// TwinCAT 3 PLC project PLC
// ProgramVersion: 3.1.4024.0
// libraries:
//   EfficientIO Communicator, * (EfficientIO)
//   EfficientIO Energy Basic, * (EfficientIO)
//   EfficientIO ModbusTCP, * (EfficientIO)
//   Lynus Energy ModbusRTU, * (Lynus AG)
//   Lynus Persistent Data V1, * (Lynus AG)
//   Lynus Standards, * (EfficientIO)
//   Tc2_Math, * (Beckhoff Automation GmbH)
//   Tc2_MBus, * (Beckhoff Automation GmbH)
//   Tc2_Standard, * (Beckhoff Automation GmbH)
//   Tc2_System, * (Beckhoff Automation GmbH)
//   Tc2_Utilities, * (Beckhoff Automation GmbH)
//   Tc3_JsonXml, * (Beckhoff Automation GmbH)
//   Tc3_Module, * (Beckhoff Automation GmbH)
// project tree:
//   / Fast_Task.TcTTO, Middle_Task.TcTTO, Slow_Task.TcTTO (not stored)
//   FB/ FB_Delta_PV_Inverter_Sunspec.TcPOU, FB_KL6xxx_ModbusRTU_22B_Master.TcPOU (not stored), FB_Shelly_3EM.TcPOU, FB_Shelly_3EM_Helper.TcPOU, FB_Shelly_HT.TcPOU (not stored), FB_Shelly_HTplus.TcPOU, FB_Shelly_HTplus_Helper.TcPOU (not stored), FB_Shelly_HT_Helper.TcPOU (not stored)
//   POUs/Backup/ prgEM.TcPOU (not stored) (excluded from build), prgEMS.TcPOU (excluded from build), prgGrid.TcPOU (excluded from build), prgHouse.TcPOU (excluded from build), prgMBUS.TcPOU (excluded from build), prgPV.TcPOU (excluded from build)
//   POUs/ MAIN.TcPOU (not stored), prgComEffIO.TcPOU, prgUv12a.TcPOU, prgPersistent.TcPOU (not stored), prgRWEffIO.TcPOU (not stored), prgVarEffIO.TcPOU (not stored)
// real-time tasks:
//   TASK Fast Task: cycle T#8ms, priority 8, ADS port 350
//   TASK Middle Task: cycle T#10ms, priority 10, ADS port 351
//   TASK Slow Task: cycle T#20ms, priority 20, ADS port 352
// I/O:
//   DEVICE Gerät 1 (Beckhoff CCAT)
//   DEVICE Gerät 2 (EtherCAT), AmsNetId 5.165.30.160.3.1
//     Klemme 1 (EK1200) [EK1200-5000 EtherCAT Netzteil (2A E-Bus)]
//       -S1 (EL2652) [EL2652 2K. Relais Ausgang, Wechsler (230V AC / 30V DC)]
//       -S2 (EL2652) [EL2652 2K. Relais Ausgang, Wechsler (230V AC / 30V DC)]
//       -S3 (EL2652) [EL2652 2K. Relais Ausgang, Wechsler (230V AC / 30V DC)]
//       -A (EL3443) [EL3443 3K. Leistungsmessung]
//       -B (EL3446) [EL3446 DPM 6 K. Strommessklemme]
//       -C (EL3446) [EL3446 DPM 6 K. Strommessklemme]
//       -D (EL3446) [EL3446 DPM 6 K. Strommessklemme]
//       Klemme 14 (EL9011) [EL9011 Endklemme]
//   DEVICE Gerät 3 (RT-Ethernet Protocol) (disabled), AmsNetId 5.165.30.160.4.1
//     BK9050 (BK9050-0000 192.168.1.118)
// variable links:
//   PLC/PLC Instance <-> Device 2 (EtherCAT)/Term 1 (EK1200)/-A (EL3443)
//     Slow_Task Inputs/prgUv12a.MessungA_ActivePower <-> Total Active/Active Power
//     Slow_Task Inputs/prgUv12a.MessungA_L1_Current <-> L1 Basic/Current
//     Slow_Task Inputs/prgUv12a.MessungA_L2_Current <-> L2 Basic/Current
//     Slow_Task Inputs/prgUv12a.MessungA_L3_Current <-> L3 Basic/Current
//     Slow_Task Inputs/prgUv12a.MessungA_L1_PowerActive <-> L1 Power/Active Power
//     Slow_Task Inputs/prgUv12a.MessungA_L2_PowerActive <-> L2 Power/Active Power
//     Slow_Task Inputs/prgUv12a.MessungA_L3_PowerActive <-> L3 Power/Active Power
//     Slow_Task Inputs/prgUv12a.MessungA_L1_PowerApparent <-> L1 Power/Apparent Power
//     Slow_Task Inputs/prgUv12a.MessungA_L2_PowerApparent <-> L2 Power/Apparent Power
//     Slow_Task Inputs/prgUv12a.MessungA_L3_PowerApparent <-> L3 Power/Apparent Power
//     Slow_Task Inputs/prgUv12a.MessungA_L1_PowerFactor <-> L1 Power/Power Factor
//     Slow_Task Inputs/prgUv12a.MessungA_L2_PowerFactor <-> L2 Power/Power Factor
//     Slow_Task Inputs/prgUv12a.MessungA_L3_PowerFactor <-> L3 Power/Power Factor
//     Slow_Task Inputs/prgUv12a.MessungA_L1_PowerReactive <-> L1 Power/Reactive Power
//     Slow_Task Inputs/prgUv12a.MessungA_L2_PowerReactive <-> L2 Power/Reactive Power
//     Slow_Task Inputs/prgUv12a.MessungA_L3_PowerReactive <-> L3 Power/Reactive Power
//     Slow_Task Inputs/prgUv12a.MessungA_L1_Voltage <-> L1 Basic/Voltage
//     Slow_Task Inputs/prgUv12a.MessungA_L2_Voltage <-> L2 Basic/Voltage
//     Slow_Task Inputs/prgUv12a.MessungA_L3_Voltage <-> L3 Basic/Voltage
//   PLC/PLC Instance <-> Device 2 (EtherCAT)/Term 1 (EK1200)/-B (EL3446)
//     Slow_Task Inputs/prgUv12a.MessungB_I{1..6}_Current <-> I{1..6} Current/Current  (6 links)
//   PLC/PLC Instance <-> Device 2 (EtherCAT)/Term 1 (EK1200)/-C (EL3446)
//     Slow_Task Inputs/prgUv12a.MessungC_I{1..6}_Current <-> I{1..6} Current/Current  (6 links)
//   PLC/PLC Instance <-> Device 2 (EtherCAT)/Term 1 (EK1200)/-D (EL3446)
//     Slow_Task Inputs/prgUv12a.MessungD_I{1..6}_Current <-> I{1..6} Current/Current  (6 links)

CONFIGURATION PLC
    RESOURCE PLC ON TwinCAT3
        TASK Fast_Task(INTERVAL := T#8ms, PRIORITY := 8);
        TASK Middle_Task(INTERVAL := T#10ms, PRIORITY := 10);
        PROGRAM prgVarEffIO WITH Fast_Task : prgVarEffIO;
        PROGRAM prgRWEffIO WITH Fast_Task : prgRWEffIO;
        PROGRAM prgPersistent WITH Middle_Task : prgPersistent;
        PROGRAM prgUv12a WITH Middle_Task : prgUv12a;
    END_RESOURCE
END_CONFIGURATION

// ---- POUs/prgUv12a.TcPOU
PROGRAM prgUv12a
// Unterverteiler 12A
VAR
{region "Daten"}
  MessungA_ActivePower      AT %I* : REAL; //{#lynus.ag#()}
  MessungA_L1_Voltage       AT %I* : REAL; //{#lynus.ag#()}
  MessungA_L1_Current       AT %I* : REAL; //{#lynus.ag#()}
  MessungA_L1_PowerActive   AT %I* : REAL; //{#lynus.ag#()}
  MessungA_L1_PowerApparent AT %I* : REAL; //{#lynus.ag#()}
  MessungA_L1_PowerReactive AT %I* : REAL; //{#lynus.ag#()}
  MessungA_L1_PowerFactor   AT %I* : REAL; //{#lynus.ag#()}
  MessungA_L2_Voltage       AT %I* : REAL; //{#lynus.ag#()}
  MessungA_L2_Current       AT %I* : REAL; //{#lynus.ag#()}
  MessungA_L2_PowerActive   AT %I* : REAL; //{#lynus.ag#()}
  MessungA_L2_PowerApparent AT %I* : REAL; //{#lynus.ag#()}
  MessungA_L2_PowerReactive AT %I* : REAL; //{#lynus.ag#()}
  MessungA_L2_PowerFactor   AT %I* : REAL; //{#lynus.ag#()}
  MessungA_L3_Voltage       AT %I* : REAL; //{#lynus.ag#()}
  MessungA_L3_Current       AT %I* : REAL; //{#lynus.ag#()}
  MessungA_L3_PowerActive   AT %I* : REAL; //{#lynus.ag#()}
  MessungA_L3_PowerApparent AT %I* : REAL; //{#lynus.ag#()}
  MessungA_L3_PowerReactive AT %I* : REAL; //{#lynus.ag#()}
  MessungA_L3_PowerFactor   AT %I* : REAL; //{#lynus.ag#()}

  MessungB_I1_Current       AT %I* : REAL; //{#lynus.ag#()}
  MessungB_I2_Current       AT %I* : REAL; //{#lynus.ag#()}
  MessungB_I3_Current       AT %I* : REAL; //{#lynus.ag#()}
  MessungB_I4_Current       AT %I* : REAL; //{#lynus.ag#()}
  MessungB_I5_Current       AT %I* : REAL; //{#lynus.ag#()}
  MessungB_I6_Current       AT %I* : REAL; //{#lynus.ag#()}

  MessungC_I1_Current       AT %I* : REAL; //{#lynus.ag#()}
  MessungC_I2_Current       AT %I* : REAL; //{#lynus.ag#()}
  MessungC_I3_Current       AT %I* : REAL; //{#lynus.ag#()}
  MessungC_I4_Current       AT %I* : REAL; //{#lynus.ag#()}
  MessungC_I5_Current       AT %I* : REAL; //{#lynus.ag#()}
  MessungC_I6_Current       AT %I* : REAL; //{#lynus.ag#()}

  MessungD_I1_Current       AT %I* : REAL; //{#lynus.ag#()}
  MessungD_I2_Current       AT %I* : REAL; //{#lynus.ag#()}
  MessungD_I3_Current       AT %I* : REAL; //{#lynus.ag#()}
  MessungD_I4_Current       AT %I* : REAL; //{#lynus.ag#()}
  MessungD_I5_Current       AT %I* : REAL; //{#lynus.ag#()}
  MessungD_I6_Current       AT %I* : REAL; //{#lynus.ag#()}
{endregion}

{region "IO"}
{endregion}
END_VAR


;

END_PROGRAM

// ---- FB/FB_Delta_PV_Inverter_Sunspec.TcPOU
FUNCTION_BLOCK FB_Delta_PV_Inverter_Sunspec
VAR_INPUT PERSISTENT
	bEnable										: BOOL;																			//{#lynus.ag#()} //Enable the Fuctionblock and his logic
	byMBAdress									: BYTE;																			//The Modbus Adress from the Slave
	diNrOfMBRTUMasterLine_IN					: DINT;																			//Number of the RTU Master Function on what this function can send or write data
END_VAR
VAR_OUTPUT
	stDeltaInverterData							: ST_DeltaPvInverter_Data;														//Structure with specific Delta Inverter Data
	stDataEMPower_PV							: ST_ElectricMeter_Output_Power;												//Output structure with Data from Electric Meter PV (Power Data)
	stDataEMCounter_PV							: ST_ElectricMeter_Output_Counter;												//Output structure with Data from Electric Meter PV (Counter Data)
	diNrOfEM_OUT_PV								: DINT;																			//Active Number from the Electric Meter for using on other functions
END_VAR
VAR
	{attribute 'hide'}
	fbElMeter									: FB_ElectricMeter;																//Electric Meter Function 
	{attribute 'hide'}
	fbNumberDevice								: FB_NumberOfDevice;															//Function block to calcualte the number of the Device
	{attribute 'hide'}
	timDelay									: TON;																			//Timer for Delay between Requests
	{attribute 'hide'}
	timTimeout									: TON;																			//Timer for Timeout
	{attribute 'hide'}
	timDissableFunctions						: TON;																			//Timer to dissable the Function after Lynus_Standards.Constants_General.tTimeDissableLynusFunctions Days without connection to the Lynus Cloud
	{attribute 'hide'}
	timResetConnectionOnGVL						: TON;																			//Timer to try reset the connection Flag on the GVL. (When somebody delete the Connection Function and make only a onlinechange)
	{attribute 'hide'}
	FPErrorMaster								: R_TRIG;																		//Internal positive Edge
	{attribute 'hide'}
	FPEnable									: R_TRIG;																		//Internal positive Edge
	{attribute 'hide'}
	fbConvertWord								: FB_CV_WORD_TO_DWORD;															//Convert 2 WORD in a DWORD
	{attribute 'hide'}
	arrPD										: ARRAY[1..5] OF FB_PersistentData_Number;										//Function to save persistent data
	{attribute 'hide'}
	arrDefaultModbusAdress						: ARRAY[1..247] OF BYTE;														//Default Modbuss Adress Array to fill in in the GVL Array after a Online change
	{attribute 'hide'}
	arrDefaultReadWrite							: ARRAY[1..Constants_Bussystems.wQuantityOfRegistersMBRTUMaster] OF WORD;		//Default Read/Write Array to fill in in the GVL Array after a Online change
	{attribute 'hide'}
	arrCounterForGVL							: ARRAY[1..2] OF DINT;															//Counter to clean old data on GVL
	{attribute 'hide'}
	bAdressIsSet								: BOOL;																			//Its true when the new Modbus Adress from the Slave is set in the Array on the GVL for the Master	
	{attribute 'hide'}
	bErrorInverter								: BOOL;																			//Error or Fault from Inverter
	{attribute 'hide'}
	bWarningInverter							: BOOL;																			//Warning from Inverter
	{attribute 'hide'}
	byWaitInStep								: BYTE;																			//Wait in Step before start to clean data on PLC
	{attribute 'hide'}
	byNumberOfSameMBAdress						: BYTE;																			//Number of Same Modbus adress on 1 Modbus Master
	{attribute 'hide'}
	byMBAdress_Old								: BYTE;																			//Old Modbus Adress to compare with the new Modbus Adress to start the state machine to set in the Array on the GVL
	{attribute 'hide'}
	byMBAdress_CP								: BYTE;																			//Variable to compare the Modbus Adress in the State Machine. When the Adress change when the state machine is active then the state machine starts from new with the new adress 
	{attribute 'hide'}
	byLPSlaveAdress								: BYTE;																			//Loop for the state machine to set the adress from the Slave in the array on the GVL
	{attribute 'hide'}
	byLPFillDefaultData							: BYTE;																			//Variable for Loop to fill default values in the Delta output structure
	{attribute 'hide'}
	byLPVendor64062								: BYTE;																			//Variable for Loop to fill the Error,Warning and Faults from Vendor 64062 to the Delta output structure
	{attribute 'hide'}
	iStateGVLData								: INT;																			//State machine to handle the data on the GVL
	{attribute 'hide'}
	iStateModbusRead							: INT;																			//State machine for read out Data over Modbus RTU
	{attribute 'hide'}
	iStateModbusError							: INT;																			//State machine for error out Data over Modbus RTU	
	{attribute 'hide'}
	iStateModbus_CP								: INT;																			//Variable to compare the state machine variable to set or reset the timeout timer
	{attribute 'hide'}
	iSFPowerMPPT								: INT;																			//Scale Factor for MPPT Power
	{attribute 'hide'}
	wNumberOfMPPT								: WORD;																			//Number of MPPT
	{attribute 'hide'}
	wLPCleanBuffer								: WORD;																			//Loop to clear the send and write Buffer on the GVL
	{attribute 'hide'}
	wLPPowerMPPT								: WORD;																			//Variable for Loop to fill the power for each MPPT in the output structure
	{attribute 'hide'}
	wNextModbusStartAdress						: WORD;																			//Next Modbus Start Adress why in Pic 160 the Number of Registers is variabel and so the next Modbus Registers in the next Pics can be different
	{attribute 'hide'}
	wNumberOfInputs								: WORD;																			//Number of Inputs from Pic 401 to calculate the Next Modbus Start Adress
	{attribute 'hide'}
	wPicID										: WORD;																			//ID of the PIC
	{attribute 'hide'}
	diNrOfMBRTUMasterLine_IN_Old				: DINT;																			//Old Modbus RTU Line to compare with the new Modbus RTU Line to start the state machine to set in the Array on the GVL
	{attribute 'hide'}
	diNrOfMBRTUMasterLine_IN_CP					: DINT;																			//Variable to compare the Modbus RTU Line in the State Machine. When the Modbus RTU Line change when the state machine is active then the state machine starts from new with the new Modbus RTU Line
	{attribute 'hide'}
	lrRestNextAdress							: LREAL;																		//Rest of the calculation for new Star Adress. In Sunspec each new PIC start with a even adress
END_VAR
VAR PERSISTENT
	{attribute 'conditionalshow'}
	byMBAdress_ForChange						: BYTE;																			//When we have 2 same Adresses on 1 Modbus RTU Line the byMBAdress_Int is set to 0. After a other change on the Input Adress Field so we can start to set the Adress in the Array in the GVL
	byMBAdress_Int								: BYTE;																			//Internal Adress what is using for the Read and Write functions
END_VAR

//Creator : Kai Ebensperger
//Company : Lynus AG
//Date : 26.10.2021
//Version : 1.0.0.0

//With this function its possible to read out values from the Delta PV Inverter over Modbus RTU
//The Protocoll is the Sunspec Protocol
//Versions that are supported : 1.16
//This Function use the INT+Scalfactor Format

//Infos for Operating State


//NOTE for diNr.....Designation => 
//_IN = Here Data come in from other Functions or go out to other functions about the GVL
//_OUT = Here Data go out to other functions about the GVL

(*--------------------------------------------------------------------------------------------Limits-------------------------------------------------------------------------------------*)

byMBAdress := LIMIT(0,byMBAdress,247);
	diNrOfMBRTUMasterLine_IN := LIMIT(0,diNrOfMBRTUMasterLine_IN,Constants_Bussystems.diMaxNumberOfMBRTUMasterKL6xxx);	

(*-------------------------------------------------------------Calcualte the number of ECS---------------------------------------------------------------*)

fbNumberDevice(
	diActualNumberOfDevices:= Lynus_Standards.GVL_Energy.stNumberOfDevices.diNumberOfElectricMeters, 
	diMaxNumberOfDevices:= Constants_Energy.diMaxNumberOfElectricMeters, 
	udiCounterOnlineChange:= TwinCAT_SystemInfoVarList._AppInfo.OnlineChangeCnt, 
	bNumberIsCalculatet=> , 
	bFPNumberIsCalculatet=> , 
	bOnlineChange=> , 
	diNumberForThisDevice=> diNrOfEM_OUT_PV, 
	diNumberOfTotalDevices=> );

//Write new Numer on GVL
IF fbNumberDevice.bFPNumberIsCalculatet THEN
	Lynus_Standards.GVL_Energy.stNumberOfDevices.diNumberOfElectricMeters := fbNumberDevice.diNumberOfTotalDevices;	
END_IF 

//Delete old Number on GVL
IF fbNumberDevice.bOnlineChange THEN 
	Lynus_Standards.GVL_Energy.stNumberOfDevices.diNumberOfElectricMeters := diNrOfEM_OUT_PV;	
		iStateGVLData := 1;	
			byMBAdress_Old := 0;
				diNrOfMBRTUMasterLine_IN_Old := 0;
END_IF

(*-------------------------------------------------------------Service from Backend is ready and check the connection to backen for dissabel/enable Function---------------------------------------------------------------*)

//Try to reset the variable for connection on the GVL. When all is normal then the Lynus Mqtt connection function set this variable to true in the next cycle
//When we have no connection to the backend then after Lynus_Standards.Constants_General.tTimeDissableLynusFunctions days the Function is dissabled with all of his functionalities
timResetConnectionOnGVL(IN:= NOT timResetConnectionOnGVL.Q, PT:= T#1H, Q=> , ET=> );
	IF timResetConnectionOnGVL.Q THEN Lynus_Standards.GVL_Communicator.bStateConnectionToEnableFunctions := FALSE; END_IF
		IF NOT Lynus_Standards.GVL_Communicator.bStateConnectionToEnableFunctions THEN timDissableFunctions.IN := TRUE; ELSE timDissableFunctions.IN := FALSE; END_IF  
			timDissableFunctions(IN:= , PT:= Lynus_Standards.Constants_General.tTimeDissableLynusFunctions, Q=> , ET=> );
			
(*--------------------------------------------------------------------------------------------Error from the Master Function-------------------------------------------------------------------------------------*)

FPErrorMaster(CLK:= Lynus_Standards.GVL_Bussystems.stDataOfMBRTUMasterKL6xxx[diNrOfMBRTUMasterLine_IN].byErrorWarning = 2 AND bEnable, Q=> );

(*--------------------------------------------------------------------------------------------Modbus Adress Slave Function-------------------------------------------------------------------------------------*)

FPEnable(CLK:= bEnable, Q=> );

//When the Adress is changed then set the new Adress in the Array
//When we have the Adress more then 1 time in 1 line then set to 0 and wait for the next change on the Input Variable for the Modbus Adress
IF byMBAdress <> byMBAdress_ForChange AND bEnable THEN byMBAdress_ForChange := byMBAdress; byNumberOfSameMBAdress := 0; END_IF     
	IF byMBAdress <> byMBAdress_Int AND byNumberOfSameMBAdress = 0 AND bEnable THEN byMBAdress_Int := byMBAdress; END_IF 
		IF NOT bEnable THEN byMBAdress_Int := 0; END_IF 
		
IF NOT Lynus_Standards.GVL_Bussystems.stDataOfMBRTUMasterKL6xxx[diNrOfMBRTUMasterLine_IN].bNoNewMBusAdress AND iStateGVLData = 0 AND (MEMCMP(ADR(byMBAdress_Int),ADR(byMBAdress_Old),SIZEOF(byMBAdress_Old)) <> 0 OR MEMCMP(ADR(diNrOfMBRTUMasterLine_IN),ADR(diNrOfMBRTUMasterLine_IN_Old),SIZEOF(diNrOfMBRTUMasterLine_IN_Old)) <> 0) THEN
	//Check if we have more then 1 time this Adress in 1 Line
	byNumberOfSameMBAdress := 0;	
		FOR byLPSlaveAdress := 1 TO 247 BY 1 DO
			IF Lynus_Standards.GVL_Bussystems.stDataOfMBRTUMasterKL6xxx[diNrOfMBRTUMasterLine_IN].arrAllModbusSlaveAdresses[byLPSlaveAdress] = byMBAdress_Int AND 
					Lynus_Standards.GVL_Bussystems.stDataOfMBRTUMasterKL6xxx[diNrOfMBRTUMasterLine_IN].arrAllModbusSlaveAdresses[byLPSlaveAdress] <> 0 THEN 
						byNumberOfSameMBAdress := byNumberOfSameMBAdress + 1; 
				END_IF 
		END_FOR
			IF byNumberOfSameMBAdress > 0 THEN 
				byMBAdress_Int := 0;
			END_IF	
				bAdressIsSet := FALSE; 
					//Delte the old Adress from the old Array
					FOR byLPSlaveAdress := 1 TO 247 BY 1 DO
						IF Lynus_Standards.GVL_Bussystems.stDataOfMBRTUMasterKL6xxx[diNrOfMBRTUMasterLine_IN_Old].arrAllModbusSlaveAdresses[byLPSlaveAdress] = byMBAdress_Old THEN
							Lynus_Standards.GVL_Bussystems.stDataOfMBRTUMasterKL6xxx[diNrOfMBRTUMasterLine_IN_Old].arrAllModbusSlaveAdresses[byLPSlaveAdress] := 0;
						END_IF	 
					END_FOR
						//Set the New Adress in Array
						byMBAdress_Old := byMBAdress_Int;
							diNrOfMBRTUMasterLine_IN_Old := diNrOfMBRTUMasterLine_IN;
								FOR byLPSlaveAdress := 1 TO 247 BY 1 DO
									IF Lynus_Standards.GVL_Bussystems.stDataOfMBRTUMasterKL6xxx[diNrOfMBRTUMasterLine_IN].arrAllModbusSlaveAdresses[byLPSlaveAdress] = 0 AND NOT bAdressIsSet THEN 
										Lynus_Standards.GVL_Bussystems.stDataOfMBRTUMasterKL6xxx[diNrOfMBRTUMasterLine_IN].arrAllModbusSlaveAdresses[byLPSlaveAdress] := byMBAdress_Int; 
											bAdressIsSet := TRUE;
									END_IF 
								END_FOR
END_IF	

(*--------------------------------------------------------------------------------------------State Machine Read--------------------------------------------------------------------------------------*)

//Timer for Delay
timDelay(IN:= , PT:= T#250MS, Q=> , ET=> );

//Timer for Timeout in Statemachine
IF iStateModbusRead > 0 AND iStateModbusRead <= 8 AND iStateModbusRead = iStateModbus_CP THEN
		timTimeout.IN := TRUE;
ELSE	
		timTimeout.IN := FALSE;
END_IF
	//Timeout Timer is dissabled when the slave wait that his adress is in porgress on the RTU Master, or is dissabled or the Terminal is not configured
	IF iStateModbusRead = 0 OR NOT bEnable OR NOT Lynus_Standards.GVL_Bussystems.stDataOfMBRTUMasterKL6xxx[diNrOfMBRTUMasterLine_IN].bTerminalIsConfigured THEN timTimeout.IN := FALSE; END_IF
		timTimeout(IN:= , PT:= T#15S, Q=> , ET=> );

//Not Enabled
IF NOT bEnable OR NOT Lynus_Standards.GVL_Bussystems.stDataOfMBRTUMasterKL6xxx[diNrOfMBRTUMasterLine_IN].bTerminalIsConfigured THEN iStateModbusRead := 0; iStateModbusError := 0; END_IF		
		
CASE iStateModbusRead OF

	0://Init Step (Wait that the Slave is enabled and the Terminal is configured)
		
		//Set Delta Output Structure to default
		IF NOT bEnable OR NOT Lynus_Standards.GVL_Bussystems.stDataOfMBRTUMasterKL6xxx[diNrOfMBRTUMasterLine_IN].bTerminalIsConfigured THEN 
			stDeltaInverterData.rTotalMPPTPower := 0;
				stDeltaInverterData.rCabinetTemp := 0;
					stDeltaInverterData.rHeatSinkTemp := 0;
						FOR byLPFillDefaultData := 1 TO 6 BY 1 DO
							stDeltaInverterData.arrMPPTPower[byLPFillDefaultData] := 0;
						END_FOR
							stDeltaInverterData.eEvent1 := eDeltaEvent.eNoInfo;
								stDeltaInverterData.eOperatingState := eDeltaOperatingState.eNoInfo;
		END_IF
		
		iSFPowerMPPT := 0;
			wNumberOfMPPT := 0;
				wNextModbusStartAdress := 0;
					wNumberOfInputs := 0;
						lrRestNextAdress := 0;
				
		IF bEnable AND Lynus_Standards.GVL_Bussystems.stDataOfMBRTUMasterKL6xxx[diNrOfMBRTUMasterLine_IN].bTerminalIsConfigured THEN
			//Start Timer for start the Statemachine
			IF NOT Lynus_Standards.GVL_Bussystems.stDataOfMBRTUMasterKL6xxx[diNrOfMBRTUMasterLine_IN].bMasterIsBusy THEN timDelay.IN := TRUE; END_IF 
		
			//Reset the Read and Write Buffer on the GVL before starting
			IF byMBAdress_Int = Lynus_Standards.GVL_Bussystems.stDataOfMBRTUMasterKL6xxx[diNrOfMBRTUMasterLine_IN].byActualMBAdressInProgrss THEN
				FOR wLPCleanBuffer := 1 TO Constants_Bussystems.wQuantityOfRegistersMBRTUMaster BY 1 DO
					Lynus_Standards.GVL_Bussystems.stDataOfMBRTUMasterKL6xxx[diNrOfMBRTUMasterLine_IN].arrReadOutData[wLPCleanBuffer] := 0;
						Lynus_Standards.GVL_Bussystems.stDataOfMBRTUMasterKL6xxx[diNrOfMBRTUMasterLine_IN].arrWriteOutData[wLPCleanBuffer] := 0;
				END_FOR
			END_IF
			
			IF timDelay.Q AND byMBAdress_Int = Lynus_Standards.GVL_Bussystems.stDataOfMBRTUMasterKL6xxx[diNrOfMBRTUMasterLine_IN].byActualMBAdressInProgrss AND NOT Lynus_Standards.GVL_Bussystems.stDataOfMBRTUMasterKL6xxx[diNrOfMBRTUMasterLine_IN].bReadWriteIsDone THEN
				timDelay.IN := FALSE;
					iStateModbusRead := 1;
						diNrOfMBRTUMasterLine_IN_CP := diNrOfMBRTUMasterLine_IN;
							byMBAdress_CP := byMBAdress_Int; 	
								Lynus_Standards.GVL_Bussystems.stDataOfMBRTUMasterKL6xxx[diNrOfMBRTUMasterLine_IN].bSlaveStartReadOrWrite := FALSE;
			END_IF
		END_IF
	
	1://Read Out Values from Pic 103 of the Sunspec Protocol (Register 40084)
		iStateModbus_CP := iStateModbusRead;
		
		Lynus_Standards.GVL_Bussystems.stDataOfMBRTUMasterKL6xxx[diNrOfMBRTUMasterLine_IN].eMBRTUReadWriteMode := E_MBRTUMaster_ReadWriteMode.eModbusRTUMaster_ReadRegs;
			Lynus_Standards.GVL_Bussystems.stDataOfMBRTUMasterKL6xxx[diNrOfMBRTUMasterLine_IN].wNumberOfRegister := 39;
				Lynus_Standards.GVL_Bussystems.stDataOfMBRTUMasterKL6xxx[diNrOfMBRTUMasterLine_IN].wModbusRegister := 40073;
		
		IF NOT Lynus_Standards.GVL_Bussystems.stDataOfMBRTUMasterKL6xxx[diNrOfMBRTUMasterLine_IN].bMasterIsBusy THEN timDelay.IN := TRUE; END_IF 

		//Copy the read out Data
		IF NOT Lynus_Standards.GVL_Bussystems.stDataOfMBRTUMasterKL6xxx[diNrOfMBRTUMasterLine_IN].bMasterIsBusy AND Lynus_Standards.GVL_Bussystems.stDataOfMBRTUMasterKL6xxx[diNrOfMBRTUMasterLine_IN].byErrorWarning = 0 AND timDelay.Q AND diNrOfMBRTUMasterLine_IN = diNrOfMBRTUMasterLine_IN_CP AND byMBAdress_Int = byMBAdress_CP THEN
			//Current L1
			IF WORD_TO_INT(Lynus_Standards.GVL_Bussystems.stDataOfMBRTUMasterKL6xxx[diNrOfMBRTUMasterLine_IN].arrReadOutData[4]) >= - 10 AND WORD_TO_INT(Lynus_Standards.GVL_Bussystems.stDataOfMBRTUMasterKL6xxx[diNrOfMBRTUMasterLine_IN].arrReadOutData[4]) <= 10 THEN
				fbElMeter.lrCurrentL1 := Lynus_Standards.GVL_Bussystems.stDataOfMBRTUMasterKL6xxx[diNrOfMBRTUMasterLine_IN].arrReadOutData[1] * EXPT(10,WORD_TO_INT(Lynus_Standards.GVL_Bussystems.stDataOfMBRTUMasterKL6xxx[diNrOfMBRTUMasterLine_IN].arrReadOutData[4]));
			END_IF
			//Current L2
			IF WORD_TO_INT(Lynus_Standards.GVL_Bussystems.stDataOfMBRTUMasterKL6xxx[diNrOfMBRTUMasterLine_IN].arrReadOutData[4]) >= - 10 AND WORD_TO_INT(Lynus_Standards.GVL_Bussystems.stDataOfMBRTUMasterKL6xxx[diNrOfMBRTUMasterLine_IN].arrReadOutData[4]) <= 10 THEN
				fbElMeter.lrCurrentL2 := Lynus_Standards.GVL_Bussystems.stDataOfMBRTUMasterKL6xxx[diNrOfMBRTUMasterLine_IN].arrReadOutData[2] * EXPT(10,WORD_TO_INT(Lynus_Standards.GVL_Bussystems.stDataOfMBRTUMasterKL6xxx[diNrOfMBRTUMasterLine_IN].arrReadOutData[4]));
			END_IF
			//Current L3
			IF WORD_TO_INT(Lynus_Standards.GVL_Bussystems.stDataOfMBRTUMasterKL6xxx[diNrOfMBRTUMasterLine_IN].arrReadOutData[4]) >= - 10 AND WORD_TO_INT(Lynus_Standards.GVL_Bussystems.stDataOfMBRTUMasterKL6xxx[diNrOfMBRTUMasterLine_IN].arrReadOutData[4]) <= 10 THEN
				fbElMeter.lrCurrentL3 := Lynus_Standards.GVL_Bussystems.stDataOfMBRTUMasterKL6xxx[diNrOfMBRTUMasterLine_IN].arrReadOutData[3] * EXPT(10,WORD_TO_INT(Lynus_Standards.GVL_Bussystems.stDataOfMBRTUMasterKL6xxx[diNrOfMBRTUMasterLine_IN].arrReadOutData[4]));
			END_IF
			//Voltage L1/N
			IF WORD_TO_INT(Lynus_Standards.GVL_Bussystems.stDataOfMBRTUMasterKL6xxx[diNrOfMBRTUMasterLine_IN].arrReadOutData[11]) >= - 10 AND WORD_TO_INT(Lynus_Standards.GVL_Bussystems.stDataOfMBRTUMasterKL6xxx[diNrOfMBRTUMasterLine_IN].arrReadOutData[11]) <= 10 THEN
				fbElMeter.lrVoltageL1N := Lynus_Standards.GVL_Bussystems.stDataOfMBRTUMasterKL6xxx[diNrOfMBRTUMasterLine_IN].arrReadOutData[8] * EXPT(10,WORD_TO_INT(Lynus_Standards.GVL_Bussystems.stDataOfMBRTUMasterKL6xxx[diNrOfMBRTUMasterLine_IN].arrReadOutData[11]));
			END_IF
			//Voltage L2/N
			IF WORD_TO_INT(Lynus_Standards.GVL_Bussystems.stDataOfMBRTUMasterKL6xxx[diNrOfMBRTUMasterLine_IN].arrReadOutData[11]) >= - 10 AND WORD_TO_INT(Lynus_Standards.GVL_Bussystems.stDataOfMBRTUMasterKL6xxx[diNrOfMBRTUMasterLine_IN].arrReadOutData[11]) <= 10 THEN
				fbElMeter.lrVoltageL2N := Lynus_Standards.GVL_Bussystems.stDataOfMBRTUMasterKL6xxx[diNrOfMBRTUMasterLine_IN].arrReadOutData[9] * EXPT(10,WORD_TO_INT(Lynus_Standards.GVL_Bussystems.stDataOfMBRTUMasterKL6xxx[diNrOfMBRTUMasterLine_IN].arrReadOutData[11]));
			END_IF
			//Voltage L3/N
			IF WORD_TO_INT(Lynus_Standards.GVL_Bussystems.stDataOfMBRTUMasterKL6xxx[diNrOfMBRTUMasterLine_IN].arrReadOutData[11]) >= - 10 AND WORD_TO_INT(Lynus_Standards.GVL_Bussystems.stDataOfMBRTUMasterKL6xxx[diNrOfMBRTUMasterLine_IN].arrReadOutData[11]) <= 10 THEN
				fbElMeter.lrVoltageL3N := Lynus_Standards.GVL_Bussystems.stDataOfMBRTUMasterKL6xxx[diNrOfMBRTUMasterLine_IN].arrReadOutData[10] * EXPT(10,WORD_TO_INT(Lynus_Standards.GVL_Bussystems.stDataOfMBRTUMasterKL6xxx[diNrOfMBRTUMasterLine_IN].arrReadOutData[11]));
			END_IF
			//AC Power
			IF WORD_TO_INT(Lynus_Standards.GVL_Bussystems.stDataOfMBRTUMasterKL6xxx[diNrOfMBRTUMasterLine_IN].arrReadOutData[13]) >= - 10 AND WORD_TO_INT(Lynus_Standards.GVL_Bussystems.stDataOfMBRTUMasterKL6xxx[diNrOfMBRTUMasterLine_IN].arrReadOutData[13]) <= 10 THEN  
				fbElMeter.lrPowerTotal := WORD_TO_INT(Lynus_Standards.GVL_Bussystems.stDataOfMBRTUMasterKL6xxx[diNrOfMBRTUMasterLine_IN].arrReadOutData[12]) * EXPT(10,WORD_TO_INT(Lynus_Standards.GVL_Bussystems.stDataOfMBRTUMasterKL6xxx[diNrOfMBRTUMasterLine_IN].arrReadOutData[13]));
			END_IF
			//Hz
			IF WORD_TO_INT(Lynus_Standards.GVL_Bussystems.stDataOfMBRTUMasterKL6xxx[diNrOfMBRTUMasterLine_IN].arrReadOutData[15]) >= - 10 AND WORD_TO_INT(Lynus_Standards.GVL_Bussystems.stDataOfMBRTUMasterKL6xxx[diNrOfMBRTUMasterLine_IN].arrReadOutData[15]) <= 10 THEN  
				fbElMeter.lrFrequency := Lynus_Standards.GVL_Bussystems.stDataOfMBRTUMasterKL6xxx[diNrOfMBRTUMasterLine_IN].arrReadOutData[14] * EXPT(10,WORD_TO_INT(Lynus_Standards.GVL_Bussystems.stDataOfMBRTUMasterKL6xxx[diNrOfMBRTUMasterLine_IN].arrReadOutData[15]));
			END_IF
			//Apparent Power
			IF WORD_TO_INT(Lynus_Standards.GVL_Bussystems.stDataOfMBRTUMasterKL6xxx[diNrOfMBRTUMasterLine_IN].arrReadOutData[17]) >= - 10 AND WORD_TO_INT(Lynus_Standards.GVL_Bussystems.stDataOfMBRTUMasterKL6xxx[diNrOfMBRTUMasterLine_IN].arrReadOutData[17]) <= 10 THEN  
				fbElMeter.lrApparentPowerTotal := WORD_TO_INT(Lynus_Standards.GVL_Bussystems.stDataOfMBRTUMasterKL6xxx[diNrOfMBRTUMasterLine_IN].arrReadOutData[16]) * EXPT(10,WORD_TO_INT(Lynus_Standards.GVL_Bussystems.stDataOfMBRTUMasterKL6xxx[diNrOfMBRTUMasterLine_IN].arrReadOutData[17]));
			END_IF
			//Reactive Power
			IF WORD_TO_INT(Lynus_Standards.GVL_Bussystems.stDataOfMBRTUMasterKL6xxx[diNrOfMBRTUMasterLine_IN].arrReadOutData[19]) >= - 10 AND WORD_TO_INT(Lynus_Standards.GVL_Bussystems.stDataOfMBRTUMasterKL6xxx[diNrOfMBRTUMasterLine_IN].arrReadOutData[19]) <= 10 THEN  
				fbElMeter.lrReactivePowerTotal := WORD_TO_INT(Lynus_Standards.GVL_Bussystems.stDataOfMBRTUMasterKL6xxx[diNrOfMBRTUMasterLine_IN].arrReadOutData[18]) * EXPT(10,WORD_TO_INT(Lynus_Standards.GVL_Bussystems.stDataOfMBRTUMasterKL6xxx[diNrOfMBRTUMasterLine_IN].arrReadOutData[19]));
			END_IF
			//Produced Energy
			IF WORD_TO_INT(Lynus_Standards.GVL_Bussystems.stDataOfMBRTUMasterKL6xxx[diNrOfMBRTUMasterLine_IN].arrReadOutData[24]) >= - 10 AND WORD_TO_INT(Lynus_Standards.GVL_Bussystems.stDataOfMBRTUMasterKL6xxx[diNrOfMBRTUMasterLine_IN].arrReadOutData[24]) <= 10 THEN  
				fbConvertWord(wInputValue_1:= Lynus_Standards.GVL_Bussystems.stDataOfMBRTUMasterKL6xxx[diNrOfMBRTUMasterLine_IN].arrReadOutData[22], wInputValue_2:= Lynus_Standards.GVL_Bussystems.stDataOfMBRTUMasterKL6xxx[diNrOfMBRTUMasterLine_IN].arrReadOutData[23], eByteOrderForConvert:= eByteOrder.eBigEndian, dwOutputValue=> );
					fbElMeter.lrCounterEnergyT1_Production := fbConvertWord.dwOutputValue * EXPT(10,WORD_TO_INT(Lynus_Standards.GVL_Bussystems.stDataOfMBRTUMasterKL6xxx[diNrOfMBRTUMasterLine_IN].arrReadOutData[24]));
						fbElMeter.lrCounterEnergyT1_Production := fbElMeter.lrCounterEnergyT1_Production / 1000;
							fbElMeter.lrTotalCounterEnergy_Production := fbElMeter.lrCounterEnergyT1_Production; 	
			END_IF
			//Cabinet Temperature
			IF WORD_TO_INT(Lynus_Standards.GVL_Bussystems.stDataOfMBRTUMasterKL6xxx[diNrOfMBRTUMasterLine_IN].arrReadOutData[35]) >= - 10 AND WORD_TO_INT(Lynus_Standards.GVL_Bussystems.stDataOfMBRTUMasterKL6xxx[diNrOfMBRTUMasterLine_IN].arrReadOutData[35]) <= 10 THEN  
				stDeltaInverterData.rCabinetTemp := LREAL_TO_REAL(WORD_TO_INT(Lynus_Standards.GVL_Bussystems.stDataOfMBRTUMasterKL6xxx[diNrOfMBRTUMasterLine_IN].arrReadOutData[31]) * EXPT(10,WORD_TO_INT(Lynus_Standards.GVL_Bussystems.stDataOfMBRTUMasterKL6xxx[diNrOfMBRTUMasterLine_IN].arrReadOutData[35])));
			END_IF
			//Heat Sink Temperature
			IF WORD_TO_INT(Lynus_Standards.GVL_Bussystems.stDataOfMBRTUMasterKL6xxx[diNrOfMBRTUMasterLine_IN].arrReadOutData[35]) >= - 10 AND WORD_TO_INT(Lynus_Standards.GVL_Bussystems.stDataOfMBRTUMasterKL6xxx[diNrOfMBRTUMasterLine_IN].arrReadOutData[35]) <= 10 THEN  
				stDeltaInverterData.rHeatSinkTemp := LREAL_TO_REAL(WORD_TO_INT(Lynus_Standards.GVL_Bussystems.stDataOfMBRTUMasterKL6xxx[diNrOfMBRTUMasterLine_IN].arrReadOutData[32]) * EXPT(10,WORD_TO_INT(Lynus_Standards.GVL_Bussystems.stDataOfMBRTUMasterKL6xxx[diNrOfMBRTUMasterLine_IN].arrReadOutData[35])));
			END_IF
			//Operating State
			stDeltaInverterData.eOperatingState := eDeltaOperatingState.eNoInfo;
			IF Lynus_Standards.GVL_Bussystems.stDataOfMBRTUMasterKL6xxx[diNrOfMBRTUMasterLine_IN].arrReadOutData[36] = 1 THEN stDeltaInverterData.eOperatingState := eDeltaOperatingState.eOff;
			ELSIF Lynus_Standards.GVL_Bussystems.stDataOfMBRTUMasterKL6xxx[diNrOfMBRTUMasterLine_IN].arrReadOutData[36] = 2 THEN stDeltaInverterData.eOperatingState := eDeltaOperatingState.eSleeping;
			ELSIF Lynus_Standards.GVL_Bussystems.stDataOfMBRTUMasterKL6xxx[diNrOfMBRTUMasterLine_IN].arrReadOutData[36] = 3 THEN stDeltaInverterData.eOperatingState := eDeltaOperatingState.eStarting;
			ELSIF Lynus_Standards.GVL_Bussystems.stDataOfMBRTUMasterKL6xxx[diNrOfMBRTUMasterLine_IN].arrReadOutData[36] = 4 THEN stDeltaInverterData.eOperatingState := eDeltaOperatingState.eMppt;
			ELSIF Lynus_Standards.GVL_Bussystems.stDataOfMBRTUMasterKL6xxx[diNrOfMBRTUMasterLine_IN].arrReadOutData[36] = 5 THEN stDeltaInverterData.eOperatingState := eDeltaOperatingState.eThrottled;
			ELSIF Lynus_Standards.GVL_Bussystems.stDataOfMBRTUMasterKL6xxx[diNrOfMBRTUMasterLine_IN].arrReadOutData[36] = 6 THEN stDeltaInverterData.eOperatingState := eDeltaOperatingState.eShuttingDown;
			ELSIF Lynus_Standards.GVL_Bussystems.stDataOfMBRTUMasterKL6xxx[diNrOfMBRTUMasterLine_IN].arrReadOutData[36] = 7 THEN stDeltaInverterData.eOperatingState := eDeltaOperatingState.eFault;
			ELSIF Lynus_Standards.GVL_Bussystems.stDataOfMBRTUMasterKL6xxx[diNrOfMBRTUMasterLine_IN].arrReadOutData[36] = 8 THEN stDeltaInverterData.eOperatingState := eDeltaOperatingState.eStandby;
			END_IF 
			//Event 1
			fbConvertWord(wInputValue_1:= Lynus_Standards.GVL_Bussystems.stDataOfMBRTUMasterKL6xxx[diNrOfMBRTUMasterLine_IN].arrReadOutData[38], wInputValue_2:= Lynus_Standards.GVL_Bussystems.stDataOfMBRTUMasterKL6xxx[diNrOfMBRTUMasterLine_IN].arrReadOutData[39], eByteOrderForConvert:= eByteOrder.eBigEndian, dwOutputValue=> );
			stDeltaInverterData.eEvent1 := eDeltaEvent.eNoInfo;
			IF fbConvertWord.dwOutputValue.0 THEN stDeltaInverterData.eEvent1 := eDeltaEvent.eGroundFault;
			ELSIF fbConvertWord.dwOutputValue.1 THEN stDeltaInverterData.eEvent1 := eDeltaEvent.eDCOverVolt;
			ELSIF fbConvertWord.dwOutputValue.2 THEN stDeltaInverterData.eEvent1 := eDeltaEvent.eACDisconnect;
			ELSIF fbConvertWord.dwOutputValue.3 THEN stDeltaInverterData.eEvent1 := eDeltaEvent.eDCDisconnect;
			ELSIF fbConvertWord.dwOutputValue.4 THEN stDeltaInverterData.eEvent1 := eDeltaEvent.eGridDisconnect;
			ELSIF fbConvertWord.dwOutputValue.5 THEN stDeltaInverterData.eEvent1 := eDeltaEvent.eCabinetOpen;
			ELSIF fbConvertWord.dwOutputValue.6 THEN stDeltaInverterData.eEvent1 := eDeltaEvent.eManualShutdown;
			ELSIF fbConvertWord.dwOutputValue.7 THEN stDeltaInverterData.eEvent1 := eDeltaEvent.eOverTemp;
			ELSIF fbConvertWord.dwOutputValue.8 THEN stDeltaInverterData.eEvent1 := eDeltaEvent.eOverFrequency;
			ELSIF fbConvertWord.dwOutputValue.9 THEN stDeltaInverterData.eEvent1 := eDeltaEvent.eUnderFrequency;
			ELSIF fbConvertWord.dwOutputValue.10 THEN stDeltaInverterData.eEvent1 := eDeltaEvent.eACOverVolt;
			ELSIF fbConvertWord.dwOutputValue.11 THEN stDeltaInverterData.eEvent1 := eDeltaEvent.eACUnderVolt;
			ELSIF fbConvertWord.dwOutputValue.12 THEN stDeltaInverterData.eEvent1 := eDeltaEvent.eBlownStringFuse;
			ELSIF fbConvertWord.dwOutputValue.13 THEN stDeltaInverterData.eEvent1 := eDeltaEvent.eUnderTemp;
			ELSIF fbConvertWord.dwOutputValue.14 THEN stDeltaInverterData.eEvent1 := eDeltaEvent.eMemoryLoss;
			ELSIF fbConvertWord.dwOutputValue.15 THEN stDeltaInverterData.eEvent1 := eDeltaEvent.eHWTestFailure;
			ELSIF fbConvertWord.dwOutputValue.16 THEN stDeltaInverterData.eEvent1 := eDeltaEvent.eOtherAlarm;
			ELSIF fbConvertWord.dwOutputValue.17 THEN stDeltaInverterData.eEvent1 := eDeltaEvent.eOtherWarning;	
			END_IF
		END_IF     				
		
		//Send the Read or Write Command to the Master
		Lynus_Standards.GVL_Bussystems.stDataOfMBRTUMasterKL6xxx[diNrOfMBRTUMasterLine_IN].bSlaveStartReadOrWrite := TRUE;
		
		//Go to the Next Step
		IF NOT Lynus_Standards.GVL_Bussystems.stDataOfMBRTUMasterKL6xxx[diNrOfMBRTUMasterLine_IN].bMasterIsBusy AND Lynus_Standards.GVL_Bussystems.stDataOfMBRTUMasterKL6xxx[diNrOfMBRTUMasterLine_IN].byErrorWarning = 0 AND timDelay.Q AND 
			diNrOfMBRTUMasterLine_IN = diNrOfMBRTUMasterLine_IN_CP AND byMBAdress_Int = byMBAdress_CP AND NOT timTimeout.Q THEN
				timDelay.IN := FALSE;
					Lynus_Standards.GVL_Bussystems.stDataOfMBRTUMasterKL6xxx[diNrOfMBRTUMasterLine_IN].bSlaveStartReadOrWrite := FALSE;
						iStateModbusRead := 2;
							wNextModbusStartAdress := 40122;		
		END_IF

			//Error on Master, changes on Inputs or Timeout
		 	IF timTimeout.Q OR diNrOfMBRTUMasterLine_IN <> diNrOfMBRTUMasterLine_IN_CP OR byMBAdress_Int <> byMBAdress_CP OR FPErrorMaster.Q THEN 
				iStateModbusError := 300; 
					diNrOfMBRTUMasterLine_IN_CP := diNrOfMBRTUMasterLine_IN; 
						byMBAdress_CP := byMBAdress_Int; 
			END_IF 
	
	2://Read Out Values from Pic 120 to Start Adress for PIC 160 of the Sunspec Protocoll		
		iStateModbus_CP := iStateModbusRead;
		
		Lynus_Standards.GVL_Bussystems.stDataOfMBRTUMasterKL6xxx[diNrOfMBRTUMasterLine_IN].eMBRTUReadWriteMode := E_MBRTUMaster_ReadWriteMode.eModbusRTUMaster_ReadRegs;
			Lynus_Standards.GVL_Bussystems.stDataOfMBRTUMasterKL6xxx[diNrOfMBRTUMasterLine_IN].wNumberOfRegister := 2;
				Lynus_Standards.GVL_Bussystems.stDataOfMBRTUMasterKL6xxx[diNrOfMBRTUMasterLine_IN].wModbusRegister := wNextModbusStartAdress;
		
		IF NOT Lynus_Standards.GVL_Bussystems.stDataOfMBRTUMasterKL6xxx[diNrOfMBRTUMasterLine_IN].bMasterIsBusy THEN timDelay.IN := TRUE; END_IF 

		//Copy the read out Data
		IF NOT Lynus_Standards.GVL_Bussystems.stDataOfMBRTUMasterKL6xxx[diNrOfMBRTUMasterLine_IN].bMasterIsBusy AND Lynus_Standards.GVL_Bussystems.stDataOfMBRTUMasterKL6xxx[diNrOfMBRTUMasterLine_IN].byErrorWarning = 0 AND timDelay.Q AND diNrOfMBRTUMasterLine_IN = diNrOfMBRTUMasterLine_IN_CP AND byMBAdress_Int = byMBAdress_CP THEN
			//PIC ID
			wPicID := Lynus_Standards.GVL_Bussystems.stDataOfMBRTUMasterKL6xxx[diNrOfMBRTUMasterLine_IN].arrReadOutData[1];
			//Number of Inputs
			wNumberOfInputs := Lynus_Standards.GVL_Bussystems.stDataOfMBRTUMasterKL6xxx[diNrOfMBRTUMasterLine_IN].arrReadOutData[2];
		END_IF     					
		
		//Send the Read or Write Command to the Master
		Lynus_Standards.GVL_Bussystems.stDataOfMBRTUMasterKL6xxx[diNrOfMBRTUMasterLine_IN].bSlaveStartReadOrWrite := TRUE;
		
		//Go to the Next Step
		IF NOT Lynus_Standards.GVL_Bussystems.stDataOfMBRTUMasterKL6xxx[diNrOfMBRTUMasterLine_IN].bMasterIsBusy AND Lynus_Standards.GVL_Bussystems.stDataOfMBRTUMasterKL6xxx[diNrOfMBRTUMasterLine_IN].byErrorWarning = 0 AND timDelay.Q AND 
			diNrOfMBRTUMasterLine_IN = diNrOfMBRTUMasterLine_IN_CP AND byMBAdress_Int = byMBAdress_CP AND NOT timTimeout.Q THEN
				timDelay.IN := FALSE;
					Lynus_Standards.GVL_Bussystems.stDataOfMBRTUMasterKL6xxx[diNrOfMBRTUMasterLine_IN].bSlaveStartReadOrWrite := FALSE;
						iStateModbusRead := 3;	
							lrRestNextAdress := 0;
			//Calculate next Modbus Start Adress for next Pic
			wNextModbusStartAdress := wNextModbusStartAdress + wNumberOfInputs + 2;
				lrRestNextAdress := FRAC(WORD_TO_REAL(wNextModbusStartAdress) / 2);	
					//If it ends with an odd number, the next PIC starts with an even address
					IF lrRestNextAdress <> 0 THEN wNextModbusStartAdress := wNextModbusStartAdress + 1; END_IF 
		END_IF

			//Error on Master, changes on Inputs or Timeout
		 	IF timTimeout.Q OR diNrOfMBRTUMasterLine_IN <> diNrOfMBRTUMasterLine_IN_CP OR byMBAdress_Int <> byMBAdress_CP OR FPErrorMaster.Q THEN 
				iStateModbusError := 300; 
					diNrOfMBRTUMasterLine_IN_CP := diNrOfMBRTUMasterLine_IN; 
						byMBAdress_CP := byMBAdress_Int; 
			END_IF		
	
	3://Check the PIC ID
		iStateModbus_CP := iStateModbusRead;
		
		IF wPicID < 160 THEN
			//Back to Step 2
			iStateModbusRead := 2;
		ELSE
			//next Step with values
			iStateModbusRead := 4;
				//Calculate next Modbus Start Adress for next Pic
				wNextModbusStartAdress := wNextModbusStartAdress - wNumberOfInputs - 2;
		END_IF
		
	
	4://Read Out Values from Pic 160 of the Sunspec Protocol
		iStateModbus_CP := iStateModbusRead;
		
		Lynus_Standards.GVL_Bussystems.stDataOfMBRTUMasterKL6xxx[diNrOfMBRTUMasterLine_IN].eMBRTUReadWriteMode := E_MBRTUMaster_ReadWriteMode.eModbusRTUMaster_ReadRegs;
			Lynus_Standards.GVL_Bussystems.stDataOfMBRTUMasterKL6xxx[diNrOfMBRTUMasterLine_IN].wNumberOfRegister := 9;
				Lynus_Standards.GVL_Bussystems.stDataOfMBRTUMasterKL6xxx[diNrOfMBRTUMasterLine_IN].wModbusRegister := wNextModbusStartAdress;
		
		IF NOT Lynus_Standards.GVL_Bussystems.stDataOfMBRTUMasterKL6xxx[diNrOfMBRTUMasterLine_IN].bMasterIsBusy THEN timDelay.IN := TRUE; END_IF 

		//Copy the read out Data
		IF NOT Lynus_Standards.GVL_Bussystems.stDataOfMBRTUMasterKL6xxx[diNrOfMBRTUMasterLine_IN].bMasterIsBusy AND Lynus_Standards.GVL_Bussystems.stDataOfMBRTUMasterKL6xxx[diNrOfMBRTUMasterLine_IN].byErrorWarning = 0 AND timDelay.Q AND diNrOfMBRTUMasterLine_IN = diNrOfMBRTUMasterLine_IN_CP AND byMBAdress_Int = byMBAdress_CP THEN
			//PIC ID
			wPicID := Lynus_Standards.GVL_Bussystems.stDataOfMBRTUMasterKL6xxx[diNrOfMBRTUMasterLine_IN].arrReadOutData[1];
			//Number of Inputs
			wNumberOfInputs := Lynus_Standards.GVL_Bussystems.stDataOfMBRTUMasterKL6xxx[diNrOfMBRTUMasterLine_IN].arrReadOutData[2];
			//Scale Factor for String Power
			iSFPowerMPPT := WORD_TO_INT(Lynus_Standards.GVL_Bussystems.stDataOfMBRTUMasterKL6xxx[diNrOfMBRTUMasterLine_IN].arrReadOutData[5]);
			//Number of MPPT Moduls
			wNumberOfMPPT := Lynus_Standards.GVL_Bussystems.stDataOfMBRTUMasterKL6xxx[diNrOfMBRTUMasterLine_IN].arrReadOutData[9];
		END_IF     				
		
		//Send the Read or Write Command to the Master
		Lynus_Standards.GVL_Bussystems.stDataOfMBRTUMasterKL6xxx[diNrOfMBRTUMasterLine_IN].bSlaveStartReadOrWrite := TRUE;
		
		//Go to the Next Step
		IF NOT Lynus_Standards.GVL_Bussystems.stDataOfMBRTUMasterKL6xxx[diNrOfMBRTUMasterLine_IN].bMasterIsBusy AND Lynus_Standards.GVL_Bussystems.stDataOfMBRTUMasterKL6xxx[diNrOfMBRTUMasterLine_IN].byErrorWarning = 0 AND timDelay.Q AND 
			diNrOfMBRTUMasterLine_IN = diNrOfMBRTUMasterLine_IN_CP AND byMBAdress_Int = byMBAdress_CP AND NOT timTimeout.Q THEN
				timDelay.IN := FALSE;
					Lynus_Standards.GVL_Bussystems.stDataOfMBRTUMasterKL6xxx[diNrOfMBRTUMasterLine_IN].bSlaveStartReadOrWrite := FALSE;
						iStateModbusRead := 5;	
							wNextModbusStartAdress := wNextModbusStartAdress + 10;	
		END_IF

			//Error on Master, changes on Inputs or Timeout
		 	IF timTimeout.Q OR diNrOfMBRTUMasterLine_IN <> diNrOfMBRTUMasterLine_IN_CP OR byMBAdress_Int <> byMBAdress_CP OR FPErrorMaster.Q THEN 
				iStateModbusError := 300; 
					diNrOfMBRTUMasterLine_IN_CP := diNrOfMBRTUMasterLine_IN; 
						byMBAdress_CP := byMBAdress_Int; 
			END_IF

	5://Read Out Values from Pic 160 of the Sunspec Protocol
		iStateModbus_CP := iStateModbusRead;
		
		wNumberOfMPPT := LIMIT(1,wNumberOfMPPT,6);
			iSFPowerMPPT := LIMIT(-10,iSFPowerMPPT,10);
		
		Lynus_Standards.GVL_Bussystems.stDataOfMBRTUMasterKL6xxx[diNrOfMBRTUMasterLine_IN].eMBRTUReadWriteMode := E_MBRTUMaster_ReadWriteMode.eModbusRTUMaster_ReadRegs;
			Lynus_Standards.GVL_Bussystems.stDataOfMBRTUMasterKL6xxx[diNrOfMBRTUMasterLine_IN].wNumberOfRegister := 20 * wNumberOfMPPT;
				Lynus_Standards.GVL_Bussystems.stDataOfMBRTUMasterKL6xxx[diNrOfMBRTUMasterLine_IN].wModbusRegister := wNextModbusStartAdress;
		
		IF NOT Lynus_Standards.GVL_Bussystems.stDataOfMBRTUMasterKL6xxx[diNrOfMBRTUMasterLine_IN].bMasterIsBusy THEN timDelay.IN := TRUE; END_IF 

		IF wNumberOfMPPT <= 1 THEN
			stDeltaInverterData.arrMPPTPower[2] := 0;
				stDeltaInverterData.arrMPPTPower[3] := 0;
					stDeltaInverterData.arrMPPTPower[4] := 0;
						stDeltaInverterData.arrMPPTPower[5] := 0;
							stDeltaInverterData.arrMPPTPower[6] := 0;
		ELSIF  wNumberOfMPPT = 2 THEN
			stDeltaInverterData.arrMPPTPower[3] := 0;
				stDeltaInverterData.arrMPPTPower[4] := 0;
					stDeltaInverterData.arrMPPTPower[5] := 0;
						stDeltaInverterData.arrMPPTPower[6] := 0;
		ELSIF  wNumberOfMPPT = 3 THEN
			stDeltaInverterData.arrMPPTPower[4] := 0;
				stDeltaInverterData.arrMPPTPower[5] := 0;
					stDeltaInverterData.arrMPPTPower[6] := 0;
		ELSIF  wNumberOfMPPT = 4 THEN
			stDeltaInverterData.arrMPPTPower[5] := 0;
				stDeltaInverterData.arrMPPTPower[6] := 0;	
		ELSIF  wNumberOfMPPT = 5 THEN
			stDeltaInverterData.arrMPPTPower[6] := 0;
		END_IF
		
		//Copy the read out Data
		IF NOT Lynus_Standards.GVL_Bussystems.stDataOfMBRTUMasterKL6xxx[diNrOfMBRTUMasterLine_IN].bMasterIsBusy AND Lynus_Standards.GVL_Bussystems.stDataOfMBRTUMasterKL6xxx[diNrOfMBRTUMasterLine_IN].byErrorWarning = 0 AND timDelay.Q AND diNrOfMBRTUMasterLine_IN = diNrOfMBRTUMasterLine_IN_CP AND byMBAdress_Int = byMBAdress_CP THEN
			//MPPT Power
			FOR wLPPowerMPPT := 1 TO (20 * wNumberOfMPPT) BY 1 DO
				IF wNumberOfMPPT >= 1 AND wLPPowerMPPT = 12 THEN stDeltaInverterData.arrMPPTPower[1] := LREAL_TO_REAL(Lynus_Standards.GVL_Bussystems.stDataOfMBRTUMasterKL6xxx[diNrOfMBRTUMasterLine_IN].arrReadOutData[wLPPowerMPPT] * EXPT(10,iSFPowerMPPT) / 1000);
				ELSIF wNumberOfMPPT >= 2 AND wLPPowerMPPT = 32 THEN stDeltaInverterData.arrMPPTPower[2] := LREAL_TO_REAL(Lynus_Standards.GVL_Bussystems.stDataOfMBRTUMasterKL6xxx[diNrOfMBRTUMasterLine_IN].arrReadOutData[wLPPowerMPPT] * EXPT(10,iSFPowerMPPT) / 1000);
				ELSIF wNumberOfMPPT >= 3 AND wLPPowerMPPT = 52 THEN stDeltaInverterData.arrMPPTPower[3] := LREAL_TO_REAL(Lynus_Standards.GVL_Bussystems.stDataOfMBRTUMasterKL6xxx[diNrOfMBRTUMasterLine_IN].arrReadOutData[wLPPowerMPPT] * EXPT(10,iSFPowerMPPT) / 1000);
				ELSIF wNumberOfMPPT >= 4 AND wLPPowerMPPT = 72 THEN stDeltaInverterData.arrMPPTPower[4] := LREAL_TO_REAL(Lynus_Standards.GVL_Bussystems.stDataOfMBRTUMasterKL6xxx[diNrOfMBRTUMasterLine_IN].arrReadOutData[wLPPowerMPPT] * EXPT(10,iSFPowerMPPT) / 1000);
				ELSIF wNumberOfMPPT >= 5 AND wLPPowerMPPT = 92 THEN stDeltaInverterData.arrMPPTPower[5] := LREAL_TO_REAL(Lynus_Standards.GVL_Bussystems.stDataOfMBRTUMasterKL6xxx[diNrOfMBRTUMasterLine_IN].arrReadOutData[wLPPowerMPPT] * EXPT(10,iSFPowerMPPT) / 1000);
				ELSIF wNumberOfMPPT >= 6 AND wLPPowerMPPT = 112 THEN stDeltaInverterData.arrMPPTPower[6] := LREAL_TO_REAL(Lynus_Standards.GVL_Bussystems.stDataOfMBRTUMasterKL6xxx[diNrOfMBRTUMasterLine_IN].arrReadOutData[wLPPowerMPPT] * EXPT(10,iSFPowerMPPT) / 1000);
				END_IF     
			END_FOR 
		END_IF     				
		
		//Total DC Power
		stDeltaInverterData.rTotalMPPTPower := 0;
			FOR wLPPowerMPPT := 1 TO 6 BY 1 DO
				stDeltaInverterData.rTotalMPPTPower := stDeltaInverterData.rTotalMPPTPower + stDeltaInverterData.arrMPPTPower[wLPPowerMPPT];
			END_FOR
			
		//Send the Read or Write Command to the Master
		Lynus_Standards.GVL_Bussystems.stDataOfMBRTUMasterKL6xxx[diNrOfMBRTUMasterLine_IN].bSlaveStartReadOrWrite := TRUE;
		
		//Go to the Next Step
		IF NOT Lynus_Standards.GVL_Bussystems.stDataOfMBRTUMasterKL6xxx[diNrOfMBRTUMasterLine_IN].bMasterIsBusy AND Lynus_Standards.GVL_Bussystems.stDataOfMBRTUMasterKL6xxx[diNrOfMBRTUMasterLine_IN].byErrorWarning = 0 AND timDelay.Q AND 
			diNrOfMBRTUMasterLine_IN = diNrOfMBRTUMasterLine_IN_CP AND byMBAdress_Int = byMBAdress_CP AND NOT timTimeout.Q THEN
				timDelay.IN := FALSE;
					Lynus_Standards.GVL_Bussystems.stDataOfMBRTUMasterKL6xxx[diNrOfMBRTUMasterLine_IN].bSlaveStartReadOrWrite := FALSE;
						iStateModbusRead := 6;
							lrRestNextAdress := 0;		
			//Calculate next Modbus Start Adress for Pic 401
			wNextModbusStartAdress := wNextModbusStartAdress - 10;
				wNextModbusStartAdress := wNextModbusStartAdress + wNumberOfInputs + 2;
					lrRestNextAdress := FRAC(WORD_TO_REAL(wNextModbusStartAdress) / 2);	
						//If it ends with an odd number, the next PIC starts with an even address
						IF lrRestNextAdress <> 0 THEN wNextModbusStartAdress := wNextModbusStartAdress + 1; END_IF
		END_IF

			//Error on Master, changes on Inputs or Timeout
		 	IF timTimeout.Q OR diNrOfMBRTUMasterLine_IN <> diNrOfMBRTUMasterLine_IN_CP OR byMBAdress_Int <> byMBAdress_CP OR FPErrorMaster.Q THEN 
				iStateModbusError := 300; 
					diNrOfMBRTUMasterLine_IN_CP := diNrOfMBRTUMasterLine_IN; 
						byMBAdress_CP := byMBAdress_Int; 
			END_IF
	
	6://Read Out Values from Pic 401 to Start Adress for Vendor 64062 of the Sunspec Protocoll	
		iStateModbus_CP := iStateModbusRead;
		
		Lynus_Standards.GVL_Bussystems.stDataOfMBRTUMasterKL6xxx[diNrOfMBRTUMasterLine_IN].eMBRTUReadWriteMode := E_MBRTUMaster_ReadWriteMode.eModbusRTUMaster_ReadRegs;
			Lynus_Standards.GVL_Bussystems.stDataOfMBRTUMasterKL6xxx[diNrOfMBRTUMasterLine_IN].wNumberOfRegister := 2;
				Lynus_Standards.GVL_Bussystems.stDataOfMBRTUMasterKL6xxx[diNrOfMBRTUMasterLine_IN].wModbusRegister := wNextModbusStartAdress;
		
		IF NOT Lynus_Standards.GVL_Bussystems.stDataOfMBRTUMasterKL6xxx[diNrOfMBRTUMasterLine_IN].bMasterIsBusy THEN timDelay.IN := TRUE; END_IF 

		//Copy the read out Data
		IF NOT Lynus_Standards.GVL_Bussystems.stDataOfMBRTUMasterKL6xxx[diNrOfMBRTUMasterLine_IN].bMasterIsBusy AND Lynus_Standards.GVL_Bussystems.stDataOfMBRTUMasterKL6xxx[diNrOfMBRTUMasterLine_IN].byErrorWarning = 0 AND timDelay.Q AND diNrOfMBRTUMasterLine_IN = diNrOfMBRTUMasterLine_IN_CP AND byMBAdress_Int = byMBAdress_CP THEN
			//PIC ID
			wPicID := Lynus_Standards.GVL_Bussystems.stDataOfMBRTUMasterKL6xxx[diNrOfMBRTUMasterLine_IN].arrReadOutData[1];
			//Number of Inputs
			wNumberOfInputs := Lynus_Standards.GVL_Bussystems.stDataOfMBRTUMasterKL6xxx[diNrOfMBRTUMasterLine_IN].arrReadOutData[2];
		END_IF     					
		
		//Send the Read or Write Command to the Master
		Lynus_Standards.GVL_Bussystems.stDataOfMBRTUMasterKL6xxx[diNrOfMBRTUMasterLine_IN].bSlaveStartReadOrWrite := TRUE;
		
		//Go to the Next Step
		IF NOT Lynus_Standards.GVL_Bussystems.stDataOfMBRTUMasterKL6xxx[diNrOfMBRTUMasterLine_IN].bMasterIsBusy AND Lynus_Standards.GVL_Bussystems.stDataOfMBRTUMasterKL6xxx[diNrOfMBRTUMasterLine_IN].byErrorWarning = 0 AND timDelay.Q AND 
			diNrOfMBRTUMasterLine_IN = diNrOfMBRTUMasterLine_IN_CP AND byMBAdress_Int = byMBAdress_CP AND NOT timTimeout.Q THEN
				timDelay.IN := FALSE;
					Lynus_Standards.GVL_Bussystems.stDataOfMBRTUMasterKL6xxx[diNrOfMBRTUMasterLine_IN].bSlaveStartReadOrWrite := FALSE;
						iStateModbusRead := 7;	
							lrRestNextAdress := 0;
			//Calculate next Modbus Start Adress
			wNextModbusStartAdress := wNextModbusStartAdress + wNumberOfInputs + 2;
				lrRestNextAdress := FRAC(WORD_TO_REAL(wNextModbusStartAdress) / 2);	
					//If it ends with an odd number, the next PIC starts with an even address
					IF lrRestNextAdress <> 0 THEN wNextModbusStartAdress := wNextModbusStartAdress + 1; END_IF 
		END_IF

			//Error on Master, changes on Inputs or Timeout
		 	IF timTimeout.Q OR diNrOfMBRTUMasterLine_IN <> diNrOfMBRTUMasterLine_IN_CP OR byMBAdress_Int <> byMBAdress_CP OR FPErrorMaster.Q THEN 
				iStateModbusError := 300; 
					diNrOfMBRTUMasterLine_IN_CP := diNrOfMBRTUMasterLine_IN; 
						byMBAdress_CP := byMBAdress_Int; 
			END_IF
	
	7://Check the PIC ID
		iStateModbus_CP := iStateModbusRead;
		
		IF wPicID < 64062 THEN
			//Back to Step 6
			iStateModbusRead := 6;
		ELSE
			//next Step with values
			iStateModbusRead := 8;
				//Calculate next Modbus Start Adress for next Pic or Vendor
				wNextModbusStartAdress := wNextModbusStartAdress - wNumberOfInputs - 2;
		END_IF		
			
	8://Read Out Values from Pic Vendor 64062 of the Sunspec Protocol (Register wNextModbusStartAdress + 2)		
		iStateModbus_CP := iStateModbusRead;
		
		Lynus_Standards.GVL_Bussystems.stDataOfMBRTUMasterKL6xxx[diNrOfMBRTUMasterLine_IN].eMBRTUReadWriteMode := E_MBRTUMaster_ReadWriteMode.eModbusRTUMaster_ReadRegs;
			Lynus_Standards.GVL_Bussystems.stDataOfMBRTUMasterKL6xxx[diNrOfMBRTUMasterLine_IN].wNumberOfRegister := 16;
				Lynus_Standards.GVL_Bussystems.stDataOfMBRTUMasterKL6xxx[diNrOfMBRTUMasterLine_IN].wModbusRegister := wNextModbusStartAdress + 2;
		
		IF NOT Lynus_Standards.GVL_Bussystems.stDataOfMBRTUMasterKL6xxx[diNrOfMBRTUMasterLine_IN].bMasterIsBusy THEN timDelay.IN := TRUE; END_IF 

		//Copy the read out Data
		IF NOT Lynus_Standards.GVL_Bussystems.stDataOfMBRTUMasterKL6xxx[diNrOfMBRTUMasterLine_IN].bMasterIsBusy AND Lynus_Standards.GVL_Bussystems.stDataOfMBRTUMasterKL6xxx[diNrOfMBRTUMasterLine_IN].byErrorWarning = 0 AND timDelay.Q AND diNrOfMBRTUMasterLine_IN = diNrOfMBRTUMasterLine_IN_CP AND byMBAdress_Int = byMBAdress_CP THEN
			//Faults
			FOR byLPVendor64062 := 1 TO 8 BY 1 DO 
				stDeltaInverterData.arrCurrentFault[byLPVendor64062] := Lynus_Standards.GVL_Bussystems.stDataOfMBRTUMasterKL6xxx[diNrOfMBRTUMasterLine_IN].arrReadOutData[byLPVendor64062];
			END_FOR
			//Error
			FOR byLPVendor64062 := 9 TO 13 BY 1 DO 
				stDeltaInverterData.arrCurrentError[byLPVendor64062 - 8] := Lynus_Standards.GVL_Bussystems.stDataOfMBRTUMasterKL6xxx[diNrOfMBRTUMasterLine_IN].arrReadOutData[byLPVendor64062];
			END_FOR
			//Warning
			FOR byLPVendor64062 := 14 TO 16 BY 1 DO 
				stDeltaInverterData.arrCurrentError[byLPVendor64062 - 13] := Lynus_Standards.GVL_Bussystems.stDataOfMBRTUMasterKL6xxx[diNrOfMBRTUMasterLine_IN].arrReadOutData[byLPVendor64062];
			END_FOR
		END_IF     				
		
		//Send the Read or Write Command to the Master
		Lynus_Standards.GVL_Bussystems.stDataOfMBRTUMasterKL6xxx[diNrOfMBRTUMasterLine_IN].bSlaveStartReadOrWrite := TRUE;
		
		//Go to the Next Step
		IF NOT Lynus_Standards.GVL_Bussystems.stDataOfMBRTUMasterKL6xxx[diNrOfMBRTUMasterLine_IN].bMasterIsBusy AND Lynus_Standards.GVL_Bussystems.stDataOfMBRTUMasterKL6xxx[diNrOfMBRTUMasterLine_IN].byErrorWarning = 0 AND timDelay.Q AND 
			diNrOfMBRTUMasterLine_IN = diNrOfMBRTUMasterLine_IN_CP AND byMBAdress_Int = byMBAdress_CP AND NOT timTimeout.Q THEN
				timDelay.IN := FALSE;
					Lynus_Standards.GVL_Bussystems.stDataOfMBRTUMasterKL6xxx[diNrOfMBRTUMasterLine_IN].bSlaveStartReadOrWrite := FALSE;
						Lynus_Standards.GVL_Bussystems.stDataOfMBRTUMasterKL6xxx[diNrOfMBRTUMasterLine_IN].bReadWriteIsDone := TRUE;
							iStateModbusRead := 0;		
		END_IF

			//Error on Master, changes on Inputs or Timeout
		 	IF timTimeout.Q OR diNrOfMBRTUMasterLine_IN <> diNrOfMBRTUMasterLine_IN_CP OR byMBAdress_Int <> byMBAdress_CP OR FPErrorMaster.Q THEN 
				iStateModbusError := 300; 
					diNrOfMBRTUMasterLine_IN_CP := diNrOfMBRTUMasterLine_IN; 
						byMBAdress_CP := byMBAdress_Int; 
			END_IF
	
END_CASE

(*------------------------------------------------------------------Error and Warning----------------------------------------------------------------------------*)	

bErrorInverter := FALSE;
	bWarningInverter := FALSE;
		FOR byLPVendor64062 := 1 TO 8 BY 1 DO 
			IF stDeltaInverterData.arrCurrentFault[byLPVendor64062] <> 0 AND stDeltaInverterData.eOperatingState = eDeltaOperatingState.eFault THEN bErrorInverter := TRUE; END_IF
		END_FOR
			FOR byLPVendor64062 := 1 TO 5 BY 1 DO 
				IF stDeltaInverterData.arrCurrentError[byLPVendor64062] <> 0 AND stDeltaInverterData.eEvent1 = eDeltaEvent.eOtherAlarm THEN bErrorInverter := TRUE; END_IF
			END_FOR
				FOR byLPVendor64062 := 1 TO 3 BY 1 DO 
					IF stDeltaInverterData.arrCurrentWarning[byLPVendor64062] <> 0 AND stDeltaInverterData.eEvent1 = eDeltaEvent.eOtherWarning THEN bWarningInverter := TRUE; END_IF
				END_FOR
					IF stDeltaInverterData.eOperatingState = eDeltaOperatingState.eFault THEN bErrorInverter := TRUE; END_IF
						IF stDeltaInverterData.eEvent1 <> eDeltaEvent.eNoInfo THEN bErrorInverter := TRUE; END_IF    

IF timDissableFunctions.Q OR bWarningInverter THEN fbElMeter.bWarning := TRUE; ELSE fbElMeter.bWarning := FALSE; fbElMeter.iWarningCode := 0; END_IF   
	IF Lynus_Standards.GVL_Energy.stNumberOfDevices.diNumberOfElectricMeters > Constants_Energy.diMaxNumberOfElectricMeters OR bErrorInverter OR Lynus_Standards.GVL_Bussystems.stDataOfMBRTUMasterKL6xxx[diNrOfMBRTUMasterLine_IN].byErrorWarning = 2 OR timTimeout.Q THEN 
		fbElMeter.bError := TRUE;
	ELSE 
		fbElMeter.bError := FALSE;
			fbElMeter.iErrorCode := 0;
	END_IF

IF timDissableFunctions.Q THEN fbElMeter.iWarningCode := 0;
ELSIF bWarningInverter THEN fbElMeter.iWarningCode := 1;
END_IF    	
	
IF Lynus_Standards.GVL_Energy.stNumberOfDevices.diNumberOfElectricMeters > Constants_Energy.diMaxNumberOfElectricMeters THEN fbElMeter.iErrorCode := 1; END_IF
	IF Lynus_Standards.GVL_Bussystems.stDataOfMBRTUMasterKL6xxx[diNrOfMBRTUMasterLine_IN].byErrorWarning = 2 OR bErrorInverter OR timTimeout.Q THEN fbElMeter.iErrorCode := 0; END_IF   

(*------------------------------------------------------------------Logic----------------------------------------------------------------------------*)

//Read Out Data done for EM Function
IF iStateModbusRead <> 1 THEN fbElMeter.bReadOutDataDone := TRUE; ELSE fbElMeter.bReadOutDataDone := FALSE; END_IF

//Function block for meter data
fbElMeter(
	bEnable:= bEnable AND NOT timDissableFunctions.Q, 
	bError:= , 
	bEnableReadOutFunction:= FALSE, 
	bWriteWithDelay:= TRUE,
	bPowerDataInvers:= FALSE, 
	bReadOutDataDone:= ,
	iTimeReadOutInterval:= , 
	iErrorCode:= , 
	iWarningCode:= , 
	lrTotalCounterEnergy_Consumption:= 0, 
	lrTotalCounterEnergy_Production:= , 
	lrCounterEnergyT1_Consumption:= 0, 
	lrCounterEnergyT2_Consumption:= 0, 
	lrCounterEnergyT1_Production:= , 
	lrCounterEnergyT2_Production:= 0, 
	lrCurrentL1:= , 
	lrVoltageL1N:= , 
	lrVoltageL1L2:= , 
	lrPowerL1:= 0, 
	lrCurrentL2:= , 
	lrVoltageL2N:= , 
	lrVoltageL2L3:= , 
	lrPowerL2:= 0, 
	lrCurrentL3:= , 
	lrVoltageL3N:= , 
	lrVoltageL3L1:= , 
	lrPowerL3:= 0, 
	lrPowerTotal:= , 
	lrFrequency:= , 
	lrReactivePowerTotal:= , 
	lrApparentPowerTotal:= , 
	tTimDelayOutput:= T#5S, 
	stDataEMOutPower=> , 
	stDataEMOutPowerDelay=> stDataEMPower_PV, 
	stDataEMOutCounter=> ,
	stDataEMOutCounterDelay=> stDataEMCounter_PV, 
	bReadOutMeter=> );
	
(*------------------------------------------------------------------------------------------State Machine Error---------------------------------------------------------------------------------------------*)	

CASE iStateModbusError OF
	
	300://Error
		iStateModbus_CP := iStateModbusError;
			timDelay.IN := FALSE;
				Lynus_Standards.GVL_Bussystems.stDataOfMBRTUMasterKL6xxx[diNrOfMBRTUMasterLine_IN].bSlaveStartReadOrWrite := FALSE;
					//Restart from new with the Read out part after an Error
					iStateModbusRead := 0;	
						iStateModbusError := 0;
END_CASE

(*------------------------------------------------------------------------------------------Device Type for MB RTU Master---------------------------------------------------------------------------------------------*)	

//Send the Device Type to the Master that he can configure the Termial with the right credentials
Lynus_Standards.GVL_Bussystems.stDataOfMBRTUMasterKL6xxx[diNrOfMBRTUMasterLine_IN].eMBRTUDeviceType := E_MBRTUMaster_DeviceType.ePV_DeltaSunspec;

(*-----------------------------------------------------------Handle data to Global structure for Electric Meter system and Modbus RTU Communication-----------------------------------------------------------------*)

CASE iStateGVLData OF
	
	0://Init Step
		byWaitInStep := 0;
			arrCounterForGVL[1] := 1; arrCounterForGVL[2] := 1;
	
	1://Wait for 4 Steps before clean al Data on GVL
		byWaitInStep := byWaitInStep + 1;
			IF byWaitInStep >= 4 AND fbNumberDevice.bNumberIsCalculatet THEN iStateGVLData := 2; END_IF
				//To much Devices, back to the Init step
				IF byWaitInStep >= 4 AND NOT fbNumberDevice.bNumberIsCalculatet THEN iStateGVLData := 0; END_IF	
			
	2://Clear all Data in GVL
		Lynus_Standards.GVL_Energy.stDataElectricMeters[arrCounterForGVL[1]].bEnabled := FALSE;	
			Lynus_Standards.GVL_Energy.stDataElectricMeters[arrCounterForGVL[1]].byErrorWarning := 0;
				Lynus_Standards.GVL_Energy.stDataElectricMeters[arrCounterForGVL[1]].lrCounterEnergyT1_Consumption := 0;
					Lynus_Standards.GVL_Energy.stDataElectricMeters[arrCounterForGVL[1]].lrCounterEnergyT1_Production := 0;
						Lynus_Standards.GVL_Energy.stDataElectricMeters[arrCounterForGVL[1]].lrCounterEnergyT2_Consumption := 0;
							Lynus_Standards.GVL_Energy.stDataElectricMeters[arrCounterForGVL[1]].lrCounterEnergyT2_Production := 0;
								Lynus_Standards.GVL_Energy.stDataElectricMeters[arrCounterForGVL[1]].lrPower := 0;
									Lynus_Standards.GVL_Energy.stDataElectricMeters[arrCounterForGVL[1]].lrPowerConsumption := 0;
										Lynus_Standards.GVL_Energy.stDataElectricMeters[arrCounterForGVL[1]].lrPowerConsumption := 0;
											Lynus_Standards.GVL_Energy.stDataElectricMeters[arrCounterForGVL[1]].lrPowerProduction := 0;
												Lynus_Standards.GVL_Energy.stDataElectricMeters[arrCounterForGVL[1]].lrTotalCounterEnergy_Consumption := 0;
													Lynus_Standards.GVL_Energy.stDataElectricMeters[arrCounterForGVL[1]].lrTotalCounterEnergy_Production := 0;
		
			//Reset this Part here and not in the RTU Master because on top we write then the New Adess in the List. So in the Master we delete only the GVL after a online change what set the Master by himself
			Lynus_Standards.GVL_Bussystems.stDataOfMBRTUMasterKL6xxx[arrCounterForGVL[2]].arrAllModbusSlaveAdresses := arrDefaultModbusAdress;
				Lynus_Standards.GVL_Bussystems.stDataOfMBRTUMasterKL6xxx[arrCounterForGVL[2]].arrReadOutData := arrDefaultReadWrite;
					Lynus_Standards.GVL_Bussystems.stDataOfMBRTUMasterKL6xxx[arrCounterForGVL[2]].arrWriteOutData := arrDefaultReadWrite;
						Lynus_Standards.GVL_Bussystems.stDataOfMBRTUMasterKL6xxx[arrCounterForGVL[2]].bSlaveStartReadOrWrite := FALSE;
							Lynus_Standards.GVL_Bussystems.stDataOfMBRTUMasterKL6xxx[arrCounterForGVL[2]].eMBRTUDeviceType := E_MBRTUMaster_DeviceType.eNoModbusRTUDevice;
								Lynus_Standards.GVL_Bussystems.stDataOfMBRTUMasterKL6xxx[arrCounterForGVL[2]].eMBRTUReadWriteMode := E_MBRTUMaster_ReadWriteMode.eModbusRTUMaster_NoMode;
									Lynus_Standards.GVL_Bussystems.stDataOfMBRTUMasterKL6xxx[arrCounterForGVL[2]].wModbusRegister := 0;
										Lynus_Standards.GVL_Bussystems.stDataOfMBRTUMasterKL6xxx[arrCounterForGVL[2]].wNumberOfRegister := 0;			
		
			//Counter for MB RTU Master
			arrCounterForGVL[2] := arrCounterForGVL[2] + 1;
				arrCounterForGVL[2] := LIMIT(0,arrCounterForGVL[2],Constants_Bussystems.diMaxNumberOfMBRTUMasterKL6xxx);
			//Counter for EM
			arrCounterForGVL[1] := arrCounterForGVL[1] + 1;
				arrCounterForGVL[1] := LIMIT(0,arrCounterForGVL[1],Constants_Energy.diMaxNumberOfElectricMeters);
					//Back to the init step
					IF arrCounterForGVL[1] >= Constants_Energy.diMaxNumberOfElectricMeters AND arrCounterForGVL[2] >= Constants_Bussystems.diMaxNumberOfMBRTUMasterKL6xxx THEN iStateGVLData := 0; END_IF

END_CASE 	 

IF diNrOfEM_OUT_PV > 0 AND fbNumberDevice.bNumberIsCalculatet THEN
	Lynus_Standards.GVL_Energy.stDataElectricMeters[diNrOfEM_OUT_PV].bEnabled := fbElMeter.stDataEMOutPower.bEnabled;
		Lynus_Standards.GVL_Energy.stDataElectricMeters[diNrOfEM_OUT_PV].byErrorWarning := fbElMeter.stDataEMOutPower.byErrorWarning;
			Lynus_Standards.GVL_Energy.stDataElectricMeters[diNrOfEM_OUT_PV].lrCounterEnergyT1_Consumption := fbElMeter.stDataEMOutCounter.lrCounterEnergyT1_Consumption;
				Lynus_Standards.GVL_Energy.stDataElectricMeters[diNrOfEM_OUT_PV].lrCounterEnergyT1_Production := fbElMeter.stDataEMOutCounter.lrCounterEnergyT1_Production;
					Lynus_Standards.GVL_Energy.stDataElectricMeters[diNrOfEM_OUT_PV].lrCounterEnergyT2_Consumption := fbElMeter.stDataEMOutCounter.lrCounterEnergyT2_Consumption;
						Lynus_Standards.GVL_Energy.stDataElectricMeters[diNrOfEM_OUT_PV].lrCounterEnergyT2_Production := fbElMeter.stDataEMOutCounter.lrCounterEnergyT2_Production;		
							Lynus_Standards.GVL_Energy.stDataElectricMeters[diNrOfEM_OUT_PV].lrPower := fbElMeter.stDataEMOutPower.lrPowerTotal;
								Lynus_Standards.GVL_Energy.stDataElectricMeters[diNrOfEM_OUT_PV].lrPowerConsumption := fbElMeter.stDataEMOutPower.lrPowerConsumption;
									Lynus_Standards.GVL_Energy.stDataElectricMeters[diNrOfEM_OUT_PV].lrPowerProduction := fbElMeter.stDataEMOutPower.lrPowerProduction;
										Lynus_Standards.GVL_Energy.stDataElectricMeters[diNrOfEM_OUT_PV].lrTotalCounterEnergy_Consumption := fbElMeter.stDataEMOutCounter.lrTotalCounterEnergy_Consumption;
											Lynus_Standards.GVL_Energy.stDataElectricMeters[diNrOfEM_OUT_PV].lrTotalCounterEnergy_Production := fbElMeter.stDataEMOutCounter.lrTotalCounterEnergy_Production;
END_IF

(*----------------------------------------------------------Save persistent data----------------------------------------------------------------*)

arrPD[1](lrValue:= BOOL_TO_LREAL(bEnable), bEventBasedActive=> );
arrPD[2](lrValue:= BYTE_TO_LREAL(byMBAdress), bEventBasedActive=> );
arrPD[3](lrValue:= DINT_TO_LREAL(diNrOfMBRTUMasterLine_IN), bEventBasedActive=> );
arrPD[4](lrValue:= BYTE_TO_LREAL(byMBAdress_ForChange), bEventBasedActive=> );
arrPD[5](lrValue:= BYTE_TO_LREAL(byMBAdress_Int), bEventBasedActive=> );

END_FUNCTION_BLOCK

// ---- FB/FB_Shelly_3EM.TcPOU
FUNCTION_BLOCK FB_Shelly_3EM
VAR_INPUT
	bStart				: BOOL;
	tDelayRequest		: TIME;		//Timer for delay before start with the next read or write Request
	sHostname			: STRING(255);		//Hostname or IP Adress from the Server
END_VAR

VAR_IN_OUT
END_VAR

VAR_OUTPUT
	bValidResult		: BOOL;							//Valid Result received from Server
    bBusy				: BOOL;							//Function is Busy
    bError				: BOOL;							//Error sucess
	bDone				: BOOL;							//True after the decoding from the received Json File
	bConnected			: BOOL;							//Connection to the Server
	lrtotalpower		: LREAL;						//Received Value
	lrpowerL1			: LREAL;
	lrcurrentL1			: LREAL;
	lrvoltageL1			: LREAL;
	lrenergyL1			: LREAL;
	lrpowerL2			: LREAL;
	lrcurrentL2			: LREAL;
	lrvoltageL2			: LREAL;
	lrenergyL2			: LREAL;
	lrpowerL3			: LREAL;
	lrcurrentL3			: LREAL;
	lrvoltageL3			: LREAL;
	lrenergyL3			: LREAL;
	hrErrorCode       	: HRESULT;						//Error Result from Http Client
END_VAR

VAR
	fbClient			: FB_IotHttpClient;
	fbHttpGet			: FB_Shelly_3EM_Helper;
	timStartRequest		: TON;							//Timer to Start the Request
	FPStartRequest		: R_TRIG;						//Internal positive Edge
	FPDone				: R_TRIG;						//Internal positive Edge
	FNStart				: F_TRIG;						//Internal negative Edge
	y: INT;
END_VAR

(*------------------------------------------------------------------------------------Configure HTTP Client------------------------------------------------------------------------------------------------------*)

fbClient.sHostName := sHostname;
fbClient.tConnectionTimeout := T#30S;

IF NOT fbClient.bConfigured THEN 
	fbClient.nHostPort:= 80;
	fbClient.bKeepAlive := TRUE;
	fbClient.tConnectionTimeout := T#30S;
END_IF


//Timer to start the Request
FPStartRequest(CLK:= bStart, Q=> );
timStartRequest(IN:= fbClient.bConfigured AND bStart AND NOT timStartRequest.Q, PT:= tDelayRequest, Q=> , ET=> );

IF ((timStartRequest.Q AND NOT bBusy) OR (FPStartRequest.Q AND NOT bBusy AND fbClient.bConfigured)) THEN 
	y:=y+1;
	fbHttpGet.bSend := TRUE; 
END_IF

				
//Http Get Function
fbHttpGet(
	lrtotalpower => lrtotalpower, 
	lrpowerL1 => lrpowerL1,
	lrcurrentL1 => lrcurrentL1,
	lrvoltageL1 => lrvoltageL1,
	lrenergyL1 => lrenergyL1,
	lrpowerL2 => lrpowerL2,
	lrcurrentL2 => lrcurrentL2,
	lrvoltageL2 => lrvoltageL2,
	lrenergyL2 => lrenergyL2,
	lrpowerL3 => lrpowerL3,
	lrcurrentL3 => lrcurrentL3,
	lrvoltageL3 => lrvoltageL3,
	lrenergyL3 => lrenergyL3,
	bSend:= , 
	fbClient:= fbClient, 
	bBusy=> bBusy, 
	bError=> ,
	sContentStatus=> ,
	sContentM0=> ,
	sContentM1=> ,
	sContentM2=> );


fbHttpGet.bSend := FALSE;

FPDone(CLK:= bDone, Q=> );

(*
//Http Client
FNStart(CLK:= bStart, Q=> );
	IF FNStart.Q THEN fbClient.Disconnect(); END_IF
*)

fbClient.Execute();

//Error
IF fbHttpGet.bError OR fbClient.bError THEN 
	bError := TRUE; 
ELSE 
	bError := FALSE; 
END_IF	

hrErrorCode := fbClient.hrErrorCode;

END_FUNCTION_BLOCK

// ---- FB/FB_Shelly_3EM_Helper.TcPOU
FUNCTION_BLOCK FB_Shelly_3EM_Helper
VAR_INPUT
	bSend				: BOOL;
END_VAR

VAR_IN_OUT
	fbClient			: FB_IotHttpClient;
END_VAR

VAR_OUTPUT
	bBusy				: BOOL;
	bError				: BOOL;
	lrtotalpower		: LREAL;
	lrpowerL1			: LREAL;
	lrcurrentL1			: LREAL;
	lrvoltageL1			: LREAL;
	lrenergyL1			: LREAL;
	lrpowerL2			: LREAL;
	lrcurrentL2			: LREAL;
	lrvoltageL2			: LREAL;
	lrenergyL2			: LREAL;
	lrpowerL3			: LREAL;
	lrcurrentL3			: LREAL;
	lrvoltageL3			: LREAL;
	lrenergyL3			: LREAL;
END_VAR

VAR
	fbRequestStatus		: FB_IotHttpRequest;
	fbRequestMeter0		: FB_IotHttpRequest;
	fbRequestMeter1		: FB_IotHttpRequest;
	fbRequestMeter2		: FB_IotHttpRequest;
	fbJson				: FB_JsonDomParser;
	nState				: UDINT;
	RisingEdge			: R_TRIG;
	timTimeout			: TON;
	tTimeOut			: TIME := T#50S;
	bGetContentResult	: BOOL;
	sContentStatus		: STRING(511);
	sContentM0			: STRING(511);
	sContentM1			: STRING(511);
	sContentM2			: STRING(511);
	
	bGetJsonResult		: BOOL;
	jsonDoc				: SJsonValue;
	jsonVal				: SJsonValue;
	
	nReqCount			: UDINT;	
	nResCount			: UDINT;
	nValidResCount		: UDINT;
	nErrCount			: UDINT;
	x: INT;
END_VAR

//Timer for Timeout
timTimeout(IN:= nState = 1 AND bBusy, PT:= tTimeOut, Q=> , ET=> );
	IF timTimeout.Q THEN 
		nState := 0;
		bBusy := FALSE;
	END_IF

RisingEdge(CLK:= bSend );
CASE nState OF
0:	
	IF RisingEdge.Q THEN 
		IF 
			fbRequestStatus.SendRequest(sUri:='/status', fbClient:=fbClient, eRequestType:=ETcIotHttpRequestType.HTTP_Get, 0, 0, 0) AND
			fbRequestMeter0.SendRequest(sUri:='/emeter/0', fbClient:=fbClient, eRequestType:=ETcIotHttpRequestType.HTTP_Get, 0, 0, 0) AND 
			fbRequestMeter1.SendRequest(sUri:='/emeter/1', fbClient:=fbClient, eRequestType:=ETcIotHttpRequestType.HTTP_Get, 0, 0, 0) AND
			fbRequestMeter2.SendRequest(sUri:='/emeter/2', fbClient:=fbClient, eRequestType:=ETcIotHttpRequestType.HTTP_Get, 0, 0, 0) THEN				
			nState:= 1;
			nReqCount:= nReqCount+1;
			bBusy:= TRUE;
			bError:= FALSE;
		END_IF					
	END_IF
1:
	x:=x+1;
	IF NOT fbRequestMeter0.bBusy AND NOT fbRequestMeter1.bBusy AND NOT fbRequestMeter2.bBusy AND NOT fbRequestStatus.bBusy THEN
		bError:= TRUE;
		IF NOT fbRequestMeter0.bError THEN				 
			bGetContentResult:= fbRequestMeter0.GetContent(pContent:= ADR(sContentM0), nContentSize:= SIZEOF(sContentM0), bSetNullTermination:= TRUE);
			IF fbRequestMeter0.nStatusCode >= 200 AND fbRequestMeter0.nStatusCode < 300 THEN
				bGetJsonResult:= FALSE;
				jsonDoc:= fbRequestMeter0.GetJsonDomContent(fbJson);
				IF jsonDoc <> 0 THEN
					bGetJsonResult:= TRUE;
					IF fbJson.HasMember(jsonDoc, 'power')  THEN
						jsonVal:= fbJson.FindMember(jsonDoc, 'power');
						nValidResCount:= nValidResCount+1;
						IF fbJson.IsDouble(jsonVal) THEN							
							lrpowerL1:= fbJson.GetDouble(jsonVal);									
						END_IF
						jsonVal:= fbJson.FindMember(jsonDoc, 'current');
						nValidResCount:= nValidResCount+1;
						IF fbJson.IsDouble(jsonVal) THEN							
							lrcurrentL1:= fbJson.GetDouble(jsonVal);									
						END_IF
						jsonVal:= fbJson.FindMember(jsonDoc, 'voltage');
						nValidResCount:= nValidResCount+1;
						IF fbJson.IsDouble(jsonVal) THEN							
							lrvoltageL1:= fbJson.GetDouble(jsonVal);									
						END_IF
						jsonVal:= fbJson.FindMember(jsonDoc, 'total');
						nValidResCount:= nValidResCount+1;
						IF fbJson.IsDouble(jsonVal) THEN							
							lrenergyL1:= fbJson.GetDouble(jsonVal);									
						END_IF	
						bError:= FALSE;
						END_IF
					END_IF						
				nResCount:= nResCount+1;			
				END_IF
		END_IF
		
		IF NOT fbRequestMeter1.bError THEN				 
			bGetContentResult:= fbRequestMeter1.GetContent(pContent:= ADR(sContentM1), nContentSize:= SIZEOF(sContentM1), bSetNullTermination:= TRUE);
			IF fbRequestMeter1.nStatusCode >= 200 AND fbRequestMeter1.nStatusCode < 300 THEN
				bGetJsonResult:= FALSE;
				jsonDoc:= fbRequestMeter1.GetJsonDomContent(fbJson);
				IF jsonDoc <> 0 THEN
					bGetJsonResult:= TRUE;
					IF fbJson.HasMember(jsonDoc, 'power')  THEN
						jsonVal:= fbJson.FindMember(jsonDoc, 'power');
						nValidResCount:= nValidResCount+1;
						IF fbJson.IsDouble(jsonVal) THEN							
							lrpowerL2:= fbJson.GetDouble(jsonVal);									
						END_IF
						jsonVal:= fbJson.FindMember(jsonDoc, 'current');
						nValidResCount:= nValidResCount+1;
						IF fbJson.IsDouble(jsonVal) THEN							
							lrcurrentL2:= fbJson.GetDouble(jsonVal);									
						END_IF
						jsonVal:= fbJson.FindMember(jsonDoc, 'voltage');
						nValidResCount:= nValidResCount+1;
						IF fbJson.IsDouble(jsonVal) THEN							
							lrvoltageL2:= fbJson.GetDouble(jsonVal);									
						END_IF
						jsonVal:= fbJson.FindMember(jsonDoc, 'total');
						nValidResCount:= nValidResCount+1;
						IF fbJson.IsDouble(jsonVal) THEN							
							lrenergyL2:= fbJson.GetDouble(jsonVal);									
						END_IF	
						bError:= FALSE;
						END_IF
					END_IF						
				nResCount:= nResCount+1;			
				END_IF
		END_IF
		
		IF NOT fbRequestMeter2.bError THEN				 
			bGetContentResult:= fbRequestMeter2.GetContent(pContent:= ADR(sContentM2), nContentSize:= SIZEOF(sContentM2), bSetNullTermination:= TRUE);
			IF fbRequestMeter2.nStatusCode >= 200 AND fbRequestMeter2.nStatusCode < 300 THEN
				bGetJsonResult:= FALSE;
				jsonDoc:= fbRequestMeter2.GetJsonDomContent(fbJson);
				IF jsonDoc <> 0 THEN
					bGetJsonResult:= TRUE;
					IF fbJson.HasMember(jsonDoc, 'power')  THEN
						jsonVal:= fbJson.FindMember(jsonDoc, 'power');
						nValidResCount:= nValidResCount+1;
						IF fbJson.IsDouble(jsonVal) THEN							
							lrpowerL3:= fbJson.GetDouble(jsonVal);									
						END_IF
						jsonVal:= fbJson.FindMember(jsonDoc, 'current');
						nValidResCount:= nValidResCount+1;
						IF fbJson.IsDouble(jsonVal) THEN							
							lrcurrentL3:= fbJson.GetDouble(jsonVal);									
						END_IF
						jsonVal:= fbJson.FindMember(jsonDoc, 'voltage');
						nValidResCount:= nValidResCount+1;
						IF fbJson.IsDouble(jsonVal) THEN							
							lrvoltageL3:= fbJson.GetDouble(jsonVal);									
						END_IF
						jsonVal:= fbJson.FindMember(jsonDoc, 'total');
						nValidResCount:= nValidResCount+1;
						IF fbJson.IsDouble(jsonVal) THEN							
							lrenergyL3:= fbJson.GetDouble(jsonVal);									
						END_IF	
						bError:= FALSE;
						END_IF
					END_IF						
				nResCount:= nResCount+1;			
				END_IF
		END_IF
		
		IF NOT fbRequestStatus.bError THEN				 
			bGetContentResult:= fbRequestStatus.GetContent(pContent:= ADR(sContentStatus), nContentSize:= SIZEOF(sContentStatus), bSetNullTermination:= TRUE);
			IF fbRequestStatus.nStatusCode >= 200 AND fbRequestStatus.nStatusCode < 300 THEN
				bGetJsonResult:= FALSE;
				jsonDoc:= fbRequestStatus.GetJsonDomContent(fbJson);
				IF jsonDoc <> 0 THEN
					bGetJsonResult:= TRUE;
					IF fbJson.HasMember(jsonDoc, 'total_power')  THEN
						jsonVal:= fbJson.FindMember(jsonDoc, 'total_power');
						nValidResCount:= nValidResCount+1;
						IF fbJson.IsDouble(jsonVal) THEN							
							lrtotalpower:= fbJson.GetDouble(jsonVal);									
						END_IF
						bError:= FALSE;
					END_IF
				END_IF		
				nResCount:= nResCount+1;			
			END_IF
		END_IF
		
		nState:= 0;
		bBusy:= FALSE;
		IF bError THEN
			nErrCount:= nErrCount+1;
		END_IF
	END_IF  	
END_CASE

END_FUNCTION_BLOCK

// ---- FB/FB_Shelly_HTplus.TcPOU
FUNCTION_BLOCK FB_Shelly_HTplus
VAR_INPUT
	bStart				: BOOL;
	tDelayRequest		: TIME;		//Timer for delay before start with the next read or write Request
	sHostname			: STRING(255);		//Hostname or IP Adress from the Server
END_VAR

VAR_IN_OUT
END_VAR

VAR_OUTPUT
	bValidResult		: BOOL;							//Valid Result received from Server
    bBusy				: BOOL;							//Function is Busy
    bError				: BOOL;							//Error sucess
	bDone				: BOOL;							//True after the decoding from the received Json File
	bConnected			: BOOL;							//Connection to the Server
	lr_Temperature		: LREAL;						//Received Value
	lr_Humidity			: LREAL;
	hrErrorCode       	: HRESULT;						//Error Result from Http Client
END_VAR

VAR
	fbClient			: FB_IotHttpClient;
	fbHttpGet			: FB_Shelly_HTplus_Helper;
	timStartRequest		: TON;							//Timer to Start the Request
	FPStartRequest		: R_TRIG;						//Internal positive Edge
	FPDone				: R_TRIG;						//Internal positive Edge
	FNStart				: F_TRIG;						//Internal negative Edge
	y: INT;
END_VAR

(*------------------------------------------------------------------------------------Configure HTTP Client------------------------------------------------------------------------------------------------------*)

fbClient.sHostName := sHostname;
fbClient.tConnectionTimeout := T#30S;

IF NOT fbClient.bConfigured THEN 
	fbClient.nHostPort:= 80;
	fbClient.bKeepAlive := TRUE;
	fbClient.tConnectionTimeout := T#30S;
END_IF


//Timer to start the Request
FPStartRequest(CLK:= bStart, Q=> );
timStartRequest(IN:= fbClient.bConfigured AND bStart AND NOT timStartRequest.Q, PT:= tDelayRequest, Q=> , ET=> );

IF ((timStartRequest.Q AND NOT bBusy) OR (FPStartRequest.Q AND NOT bBusy AND fbClient.bConfigured)) THEN 
	y:=y+1;
	fbHttpGet.bSend := TRUE; 
END_IF

				
//Http Get Function

fbHttpGet(
	bSend:= , 
	fbClient:= , 
	bBusy=> , 
	bError=> , 
	lr_Temperature=> lr_Temperature, 
	lr_Humidity=> lr_Humidity,
	bSend:= , 
	fbClient:= fbClient, 
	bBusy=> bBusy, 
	bError=> ,
	sContentStatus=> ,
	sContentM0=> ,
	sContentM1=> ,
	sContentM2=> );
	



fbHttpGet.bSend := FALSE;

FPDone(CLK:= bDone, Q=> );

(*
//Http Client
FNStart(CLK:= bStart, Q=> );
	IF FNStart.Q THEN fbClient.Disconnect(); END_IF
*)

fbClient.Execute();

//Error
IF fbHttpGet.bError OR fbClient.bError THEN 
	bError := TRUE; 
ELSE 
	bError := FALSE; 
END_IF	

hrErrorCode := fbClient.hrErrorCode;

END_FUNCTION_BLOCK

// ---- POUs/Backup/prgEMS.TcPOU
PROGRAM prgEMS
VAR PERSISTENT
	byMaxDepthOfDischrgEPO		: BYTE;							//{#lynus.ag#()}
	byPrioMinChrgBattSOCInEPO	: BYTE;							//{#lynus.ag#()}
	byResChrgfromGridToBatt		: BYTE;							//{#lynus.ag#()}
	byReserveSOCEPO				: BYTE;							//{#lynus.ag#()}
	uiUpdateTime				: UINT;							//{#lynus.ag#()}
	bEnableEMS					: BOOL;							//{#lynus.ag#()}
	bAllowChrgFromGrid			: BOOL;							//{#lynus.ag#()}
	rMainFuseCSEMS				: REAL;							//{#lynus.ag#()}
	iOperationModeEMS			: INT;							//{#lynus.ag#()}
	rSizeGridConn				: REAL;							//{#lynus.ag#()}
END_VAR
VAR
	fbEMS						: FB_EMS_V2;
	bIsEnableEMS				: BOOL;							//{#lynus.ag#()}
	bStateAllowChrgFromGrid		: BOOL;							//{#lynus.ag#()}
	bStateFuseCS				: BOOL;							//{#lynus.ag#()}
	bHPActivate					: BOOL;							//{#lynus.ag#()}
	bControllingState			: BOOL;							//{#lynus.ag#()}
	iMessageEMS					: INT;							//{#lynus.ag#()}
	rHeartbeatEMS				: REAL;							//{#lynus.ag#()}
	rErrorWarningEMS			: REAL;							//{#lynus.ag#()}
	rReadyEMS					: REAL;							//{#lynus.ag#()}
	rNewBatteryPowerEMS			: REAL;							//{#lynus.ag#()}
	fbGrid: FB_Grid_Power_Ext_Input;

END_VAR

IF iOperationModeEMS = 0 THEN fbEMS.eOperationMode := E_OperatingMode_EMS.eAllOff;
ELSIF iOperationModeEMS = 1 THEN fbEMS.eOperationMode := E_OperatingMode_EMS.eSelfConsumption;	
ELSIF iOperationModeEMS = 2 THEN fbEMS.eOperationMode := E_OperatingMode_EMS.ePeakLoadCapping;
ELSIF iOperationModeEMS = 3 THEN fbEMS.eOperationMode := E_OperatingMode_EMS.eLoadManagement;			
END_IF
fbEMS.stSetupEMS.bAllowChrgFromGrid := bAllowChrgFromGrid;
fbEMS.stSetupEMS.byMaxDepthOfDischrgEPO := byMaxDepthOfDischrgEPO;
// fbEMS.stSetupEMS.byPrioMinChrgBattSOCInEPO := byPrioMinChrgBattSOCInEPO;
// fbEMS.stSetupEMS.byResChrgfromGridToBatt := byResChrgfromGridToBatt;
fbEMS.stSetupEMS.byReserveSOCEPO := byReserveSOCEPO;
//fbEMS.stSetupEMS.rSizeMainFuseCS := rMainFuseCSEMS;
fbEMS.stSizeMainFuseCS.rElSizeLine1 := rMainFuseCSEMS;
fbEMS.stSetupEMS.bEnableMainFuseFunc := bStateFuseCS;
fbEMS.stSetupEMS.uiUpdateTime := uiUpdateTime;

fbEMS(
	bEnable						:= bEnableEMS, 
//	diNrOfEM_IN_ECS				:= , 
	stSetupEMS					:= , 
	eOperationMode				:= , 
	eSpeedModeBackendController	:= E_SpeedModeBackendController_EMS.eFast, 
	eSpeedModeLocalController	:= E_SpeedModeLocalController_EMS.eFast,
	bActivateHP					:= bHPActivate, 
	bControllingState			:= bControllingState, 
	rHeartbeat					:= rHeartbeatEMS, 
	rErrorWarning				:= rErrorWarningEMS, 
	rEnergyOptReady				:= rReadyEMS, 
	rNewBattPower				:= rNewBatteryPowerEMS, 

	eMessageEMS				=> iMessageEMS, 
	bStateEnable			=> bIsEnableEMS, 
	bStateAllowChrgFromGrid	=> bStateAllowChrgFromGrid, 
	bMissingPowerData		=> , 
	bSurplusAvailable		=> , 
	byProgress				=> , 
	uiState_OUT				=> , 
	diNrOfEMS_OUT			=> , 
	arrMinPrioReached		=> , 
	arrMaxPrioReached		=> ,
	);
	
fbGrid(
	bEnable:= TRUE, 
	diNrOfEMS_IN:= prgEMS.fbEMS.diNrOfEMS_OUT, 
	rSizeGridConn:= rSizeGridConn , 
	bExtErrorGrid:= , 
	lrExtGridPower:= prgHouse.lrNetzEinspeisung , 
	lrExtTotalCounterEnergy_Consumption:= , 
	lrExtTotalCounterEnergy_Production:= , 
	lrExtCounterEnergyT1_Consumption:= , 
	lrExtCounterEnergyT2_Consumption:= , 
	lrExtCounterEnergyT1_Production:= , 
	lrExtCounterEnergyT2_Production:= , 
	stDataGrid=> , 
	diNrOfGrid_OUT=> );

END_PROGRAM

// ---- POUs/Backup/prgHouse.TcPOU
PROGRAM prgHouse
VAR
	fbKBusState					: FB_K_Bus_State;
	uint_KBusState				: UINT;							//{#lynus.ag#()}
	lrHousePower				: LREAL;								//{#lynus.ag#()}
	lrNetzEinspeisung			: LREAL;								//{#lynus.ag#()}
	lrBetriebMuellerBau			: LREAL;								//{#lynus.ag#()}
	lrElektromobilitaet			: LREAL;								//{#lynus.ag#()}
	lrHolzschnitzel				: LREAL;								//{#lynus.ag#()}
	lrLueftung_Kaelte			: LREAL;								//{#lynus.ag#()}
	//rPVProd						: REAL;									//{#lynus.ag#()}
	lrAbgaenge					: REAL;									//{#lynus.ag#()}
	fbGrid1						: FB_EM_Beckhoff_KL3403;  	//Elektromobilität 
	fbGrid2						: FB_EM_Beckhoff_KL3403;	//Holzschnitzelheizung
	fbGrid3						: FB_EM_Beckhoff_KL3403;	//Lüftung/Kälte Büro
	
	

    Volt1L1  AT %I* : REAL;
    Strom1L1 AT %I* : REAL;
	//UV Müller Holzbau
	ActivePowerTotal_1	AT %I*	: REAL;									//{#lynus.ag#()}
	//Abgang Direktmessung
	ActivePowerTotal_2	AT %I*	: REAL;									//{#lynus.ag#()}
	//Produktion PV
	ActivePowerTotal_3	AT %I*	: REAL;									//{#lynus.ag#()}

END_VAR

lrNetzEinspeisung := ActivePowerTotal_1/1000 + ActivePowerTotal_2/1000 - prgPV.PV_Gesamt;

lrElektromobilitaet	:= fbGrid1.stDataEMPower.lrPowerTotal;
lrHolzschnitzel		:= fbGrid2.stDataEMPower.lrPowerTotal;
lrLueftung_Kaelte	:= fbGrid3.stDataEMPower.lrPowerTotal;
lrHousePower		:= ActivePowerTotal_1/1000 + fbGrid1.stDataEMPower.lrPowerTotal + fbGrid2.stDataEMPower.lrPowerTotal + fbGrid3.stDataEMPower.lrPowerTotal;

lrBetriebMuellerBau := -fbGrid1.stDataEMPower.lrPowerTotal - fbGrid2.stDataEMPower.lrPowerTotal - fbGrid3.stDataEMPower.lrPowerTotal + lrHousePower;	

//rPVProd				:= (ActivePowerTotal_3)/100 * -1;					//Invertieren
lrAbgaenge 			:= ActivePowerTotal_2/1000;
//lrHousePower 		:= lrBetriebMuellerBau * -1;						//Invertierte Einspeisung für Darstellung

//The mapping of this function must be linked with the K-Bus State in the E/A Part
fbKBusState(	uiKBusState_OUT=> , 
				b_Kbus_notOk=> , 
				word_ErrorCount=> );

fbGrid1(
	bEnable:= TRUE, 
	bChannel1Invers:= FALSE, 
	bChannel2Invers:= FALSE, 
	bChannel3Invers:= FALSE, 
	uiCurrentTransformerRatioL1:= 400, 
	uiCurrentTransformerRatioL2:= 400, 
	uiCurrentTransformerRatioL3:= 400, 
	uiKBusState_IN:= fbKBusState.uiKBusState_OUT, 
	stDataEMPower=> , 
	stDataEMCounter=> , 
	stDataEMPowerRealTime=> , 
	stDataEMCounterRealTime=> , 
	diNrOfEM_OUT=> );
	
	
fbGrid2(
	bEnable:= TRUE, 
	bChannel1Invers:= FALSE, 
	bChannel2Invers:= FALSE, 
	bChannel3Invers:= FALSE, 
	uiCurrentTransformerRatioL1:= 400, 
	uiCurrentTransformerRatioL2:= 400, 
	uiCurrentTransformerRatioL3:= 400, 
	uiKBusState_IN:= , 
	stDataEMPower=> , 
	stDataEMCounter=> , 
	stDataEMPowerRealTime=> , 
	stDataEMCounterRealTime=> , 
	diNrOfEM_OUT=> );
	
fbGrid3(
	bEnable:= TRUE, 
	bChannel1Invers:= FALSE, 
	bChannel2Invers:= FALSE, 
	bChannel3Invers:= FALSE, 
	uiCurrentTransformerRatioL1:= 400, 
	uiCurrentTransformerRatioL2:= 400, 
	uiCurrentTransformerRatioL3:= 400, 
	uiKBusState_IN:= , 
	stDataEMPower=> , 
	stDataEMCounter=> , 
	stDataEMPowerRealTime=> , 
	stDataEMCounterRealTime=> , 
	diNrOfEM_OUT=> );

END_PROGRAM

// ---- POUs/Backup/prgPV.TcPOU
PROGRAM prgPV
VAR
	//fbPV1							:FB_SunSpec_PV_Inverter;
	Wechselrichter1kWRaw AT %MW0	:INT;
	Wechselrichter1kW				:REAL;							//{#lynus.ag#()}
	Wechselrichter2kWRaw AT %MW2	:INT;
	Wechselrichter2kW				:REAL;							//{#lynus.ag#()}
	Wechselrichter3kWRaw AT %MW4	:INT;
	Wechselrichter3kW				:REAL;							//{#lynus.ag#()}
	Wechselrichter4kWRaw AT %MW6	:INT;
	Wechselrichter4kW				:REAL;							//{#lynus.ag#()}
	Wechselrichter5kWRaw AT %MW8	:INT;
	Wechselrichter5kW				:REAL;							//{#lynus.ag#()}
	Wechselrichter6kWRaw AT %MW10	:INT;
	Wechselrichter6kW				:REAL;							//{#lynus.ag#()}
	Wechselrichter7kWRaw AT %MW12	:INT;
	Wechselrichter7kW				:REAL;							//{#lynus.ag#()}
	Wechselrichter8kWRaw AT %MW14	:INT;
	Wechselrichter8kW				:REAL;							//{#lynus.ag#()}
	Wechselrichter9kWRaw AT %MW16	:INT;
	Wechselrichter9kW				:REAL;							//{#lynus.ag#()}
	PV_Gesamt						:REAL;							//{#lynus.ag#()}

END_VAR

Wechselrichter1kW := TO_REAL(Wechselrichter1kWRaw) / 100.0;
Wechselrichter2kW := TO_REAL(Wechselrichter2kWRaw) / 100.0;
Wechselrichter3kW := TO_REAL(Wechselrichter3kWRaw) / 100.0;
Wechselrichter4kW := TO_REAL(Wechselrichter4kWRaw) / 100.0;
Wechselrichter5kW := TO_REAL(Wechselrichter5kWRaw) / 100.0;
Wechselrichter6kW := TO_REAL(Wechselrichter6kWRaw) / 100.0;
Wechselrichter7kW := TO_REAL(Wechselrichter7kWRaw) / 100.0;
Wechselrichter8kW := TO_REAL(Wechselrichter8kWRaw) / 100.0;
Wechselrichter9kW := TO_REAL(Wechselrichter9kWRaw) / 100.0;

PV_Gesamt 		  := Wechselrichter1kW + Wechselrichter2kW + Wechselrichter3kW + Wechselrichter4kW + Wechselrichter5kW + Wechselrichter6kW + Wechselrichter7kW + Wechselrichter8kW + Wechselrichter9kW;

(*
fbPV1(
	bEnable:= , 
	sIPAdress:= '192.168.140.6', 
	byUnitID_Inverter:= 1, 
	stDataSunSpec=> , 
	stDataEMPower_PV=> , 
	stDataEMCounter_PV=> , 
	diNrOfEM_OUT_PV=> 
);
*)

END_PROGRAM

// ---- POUs/Backup/prgGrid.TcPOU
PROGRAM prgGrid
VAR
	fbKBusState					: FB_K_Bus_State;
	fbGrid						: FB_EM_Beckhoff_KL3403;
	uint_KBusState				: UINT;							//{#lynus.ag#()}
	fbGridCounter				: FB_EnergyCounter;
	lrGridPower					: LREAL;								//{#lynus.ag#()}
	lrVoltage_L1N					: LREAL;								//{#lynus.ag#()}
	lrVoltage_L2N					: LREAL;								//{#lynus.ag#()}
	lrVoltage_L3N					: LREAL;								//{#lynus.ag#()}
END_VAR
VAR PERSISTENT
	rSizeGridConn				: REAL;									//{#lynus.ag#()}
	lrCounterGridProd			: LREAL;								//{#lynus.ag#()}
	lrCounterGridCons			: LREAL;								//{#lynus.ag#()}
END_VAR

//The mapping of this function must be linked with the K-Bus State in the E/A Part
fbKBusState(	uiKBusState_OUT=> , 
				b_Kbus_notOk=> , 
				word_ErrorCount=> );

//The mapping of this function must be linked with the KL3403 in the E/A Part
//UV1
fbGrid(
	bEnable:= TRUE, 
	bChannel1Invers:= FALSE,				//Invert power data when transformer are mounted upside down
	bChannel2Invers:= FALSE,			// CT seems to be wired the wrong wy around
	bChannel3Invers:= FALSE,
	uiCurrentTransformerRatioL1:= 400, //Transformer ratio on the secondary side
	uiCurrentTransformerRatioL2:= 400, 
	uiCurrentTransformerRatioL3:= 400, 
	uiKBusState_IN:= fbKBusState.uiKBusState_OUT, 
	stDataEMPower=> , 
	stDataEMCounter=> , 
	stDataEMPowerRealTime=> , 
	stDataEMCounterRealTime=> , 
	diNrOfEM_OUT=> );
	
uint_KBusState :=	fbKBusState.uiKBusState_OUT;
lrGridPower := fbGrid.stDataEMPower.lrPowerTotal;

// EnergyCounter
fbGridCounter(
	byActiveTariff:= 1, 
	lrPowerInput:= lrGridPower, 
	lrTotalCounterEnergy_Consumption=> , 
	lrTotalCounterEnergy_Production=> , 
	lrCounterEnergyT1_Consumption=> , 
	lrCounterEnergyT2_Consumption=> , 
	lrCounterEnergyT1_Production=> , 
	lrCounterEnergyT2_Production=> );

IF fbGridCounter.lrTotalCounterEnergy_Production > lrCounterGridProd THEN  	
		lrCounterGridProd := fbGridCounter.lrTotalCounterEnergy_Production;
END_IF

IF fbGridCounter.lrTotalCounterEnergy_Consumption > lrCounterGridCons THEN  	
	lrCounterGridCons := fbGridCounter.lrTotalCounterEnergy_Consumption;
END_IF

lrVoltage_L1N := fbGrid.stDataEMPower.lrVoltageL1N;
lrVoltage_L2N := fbGrid.stDataEMPower.lrVoltageL2N;
lrVoltage_L3N := fbGrid.stDataEMPower.lrVoltageL3N;

END_PROGRAM

// ---- POUs/Backup/prgMBUS.TcPOU
PROGRAM prgMBUS
VAR
	// M-Bus Kommunikation (KL6781)
	fbMBusKL6781         : FB_MBUSKL6781;             // Hauptbaustein für die M-Bus-Kommunikation
	stComIn              AT %I* : ST_KL6781inData22B; // Eingabestruktur für KL6781
	stComOut             AT %Q* : ST_KL6781outData22B;// Ausgabestruktur für KL6781
	stCom                : ST_MBUS_Communication;     // Kommunikationsstruktur für alle M-Bus-Geräte
	fbScann              : FB_MBUS_Scan;
	// Wärmezähler (Supercal 531)
	fbHolzkessel         : FB_MBUS_General;          	 // Funktionsbaustein für Holzkessel
	fbFussbodenheizung   : FB_MBUS_General;   		 	 // Funktionsbaustein für MAB Fußbodenheizung
	fbDSP_Produktion     : FB_MBUS_General;   			// Funktionsbaustein für DSP Produktion
	fbHeizkoerper_buero  : FB_MBUS_General;   			// Funktionsbaustein für Heizkörper Büro
	fbHalle_Bestand_S100 : FB_MBUS_General;   			// Funktionsbaustein für Halle Bestand S100
	fbLueftung	         : FB_MBUS_General;   			// Funktionsbaustein für Lüftung

	// Variablen für Steuerung
	m_Start1             : BOOL;                      
	m_Start2             : BOOL;                      
	m_Start3             : BOOL;
	m_Start4             : BOOL;
	m_Start5             : BOOL;
	m_Start6             : BOOL;
	
	//
	//TODO austausch FLOW mit Vorlauf und Rücklauftemperatur
	//
	
	// Ausgelesene Werte Wärmezähler
	lrEnergy_Holzkessel	 		: LREAL;								//{#lynus.ag#()}
	rFlow_Holzkessel     		: REAL;
	rPower_Holzkessel    		: REAL;									//{#lynus.ag#()}
	rflow_VL_Holzkessel			: REAL;									//{#lynus.ag#()}
	rflow_RL_Holzkessel			: REAL;									//{#lynus.ag#()}

	lrEnergy_Fussboden   		: LREAL;								//{#lynus.ag#()}
	rFlow_Fussboden         	: REAL;
	rPower_Fussboden        	: REAL;									//{#lynus.ag#()}
	rflow_VL_Fussboden			: REAL;									//{#lynus.ag#()}
	rflow_RL_Fussboden			: REAL;									//{#lynus.ag#()}

	lrEnergy_DSP_Produktion 	: LREAL;								//{#lynus.ag#()}
	rFlow_DSP_Produktion    	: REAL;
	rPower_DSP_Produktion   	: REAL;									//{#lynus.ag#()}
	rflow_VL_DSP_Produktion		: REAL;									//{#lynus.ag#()}
	rflow_RL_DSP_Produktion		: REAL;									//{#lynus.ag#()}
	
	lrEnergy_Heizkoerper_buero  : LREAL;								//{#lynus.ag#()}
	rFlow_Heizkoerper_buero     : REAL;
	rPower_Heizkoerper_buero    : REAL;									//{#lynus.ag#()}
	rflow_VL_Heizkoerper_buero	: REAL;									//{#lynus.ag#()}
	rflow_RL_Heizkoerper_buero	: REAL;									//{#lynus.ag#()}
	
	lrEnergy_Halle_Bestand_S100 : LREAL;								//{#lynus.ag#()}
	rFlow_Halle_Bestand_S100    : REAL;
	rPower_Halle_Bestand_S100   : REAL;									//{#lynus.ag#()}
	rflow_VL_Halle_Bestand_S100	: REAL;									//{#lynus.ag#()}
	rflow_RL_Halle_Bestand_S100	: REAL;									//{#lynus.ag#()}
	
	lrEnergy_Lueftung           : LREAL;								//{#lynus.ag#()}
	rFlow_Lueftung              : REAL;
	rPower_Lueftung             : REAL;									//{#lynus.ag#()}
	rflow_VL_Lueftung			: REAL;									//{#lynus.ag#()}
	rflow_RL_Lueftung			: REAL;									//{#lynus.ag#()}

	Err1 : E_MBUS_ERROR;
	Err2 : E_MBUS_ERROR;
	Err3 : E_MBUS_ERROR;
	Err4 : E_MBUS_ERROR;
	Err5 : E_MBUS_ERROR;
	Err6 : E_MBUS_ERROR;
	
	Busy1Trig : R_TRIG;
	DataReadyCount : DINT;
	DevError : ST_MBus_Info; 

	DataReadyCount2 : DINT;
	DevError2       : ST_MBus_Info; 

END_VAR

// ** M-Bus Hauptkommunikation **

fbMBusKL6781(
	usiRetries := 3,                    // Anzahl der Wiederholungen bei Fehler
	bStart := TRUE,                     // Startet die M-Bus-Kommunikation
	bDisabled := FALSE,                 // Deaktiviert die M-Bus-Kommunikation nicht
	bBusy => , 
	bReady => , 
	bError => , 
	eError => , 
	stComIn := stComIn, 
	stComOut := stComOut, 
	stCom := stCom
);

fbScann(
	bStart:= , 
	bStop:= , 
	eBaudrate:= E_MBUS_Baudrate.eMBus_Baud2400, 
	bDisabled:= , 
	bBusy=> , 
	bReady=> , 
	bError=> , 
	eError=> , 
	usiAddress=> , 
	usiCount=> , 
	arrDevice=> , 
	stCom:= stCom);


// ** Holzkessel (Supercal 531) auslesen **

//fbSupercal1.stSecAdr.udiIdNumber:= 30868639;

fbHolzkessel(
	usiAddress 	:= 1,                    	// M-Bus-Adresse(Primär)
	bStart 		:= m_Start1,                // Startflag
	usiUnit     := 1,               		// KW
	bDisabled 	:= FALSE,                 	
	bBusy => , 
	bReady => ,              				// Datenbereit-Status
	bError => , 
	eError => , 
	stCom 		:= stCom
);

IF NOT fbHolzkessel.bBusy AND fbHolzkessel.bError THEN

	Err1:= fbHolzkessel.eError;
END_IF

IF fbHolzkessel.bReady THEN

    lrEnergy_Holzkessel 	:= STRING_TO_REAL(fbHolzkessel.arrData[1].sValue);                 	// Energie (kWh)
    rFlow_Holzkessel 		:= STRING_TO_REAL(fbHolzkessel.arrData[6].sValue);                  // Durchfluss (m³/h)
    rPower_Holzkessel 	:= STRING_TO_REAL(fbHolzkessel.arrData[7].sValue);                    	// Leistung (kW)
END_IF

fbFussbodenheizung(
	usiAddress 	:= 2,                    	// M-Bus-Adresse(Primär)
	bStart 		:= m_Start2,                // Startflag
	usiUnit     := 1,               		// KW
	bDisabled 	:= FALSE,                 	
	bBusy => , 
	bReady => ,              				// Datenbereit-Status
	bError => , 
	eError => , 
	stCom 		:= stCom
);

IF NOT fbFussbodenheizung.bBusy AND fbFussbodenheizung.bError THEN

	Err2:= fbFussbodenheizung.eError;
END_IF

IF fbFussbodenheizung.bReady THEN

    lrEnergy_Fussboden 	:= STRING_TO_REAL(fbFussbodenheizung.arrData[1].sValue);                // Energie (kWh)
    rFlow_Fussboden 	:= STRING_TO_REAL(fbFussbodenheizung.arrData[6].sValue);                // Durchfluss (m³/h)
    rPower_Fussboden 	:= STRING_TO_REAL(fbFussbodenheizung.arrData[7].sValue);                // Leistung (kW)
	rflow_VL_Fussboden	:= STRING_TO_REAL(fbFussbodenheizung.arrData[3].sValue);					// Temperatur in Grad C
	rflow_RL_Fussboden	:= STRING_TO_REAL(fbFussbodenheizung.arrData[4].sValue);					// Temperatur in Grad C
END_IF

fbDSP_Produktion(
	usiAddress 	:= 3,                    	// M-Bus-Adresse(Primär)
	bStart 		:= m_Start3,                // Startflag
	usiUnit     := 1,               		// KW
	bDisabled 	:= FALSE,                 	
	bBusy => , 
	bReady => ,              				// Datenbereit-Status
	bError => , 
	eError => , 
	stCom 		:= stCom
);

IF NOT fbDSP_Produktion.bBusy AND fbDSP_Produktion.bError THEN

	Err3:= fbDSP_Produktion.eError;
END_IF

IF fbDSP_Produktion.bReady THEN

    lrEnergy_DSP_Produktion 	:= STRING_TO_REAL(fbDSP_Produktion.arrData[1].sValue);                 	// Energie (kWh)
    rFlow_DSP_Produktion 		:= STRING_TO_REAL(fbDSP_Produktion.arrData[6].sValue);                  // Durchfluss (m³/h)
    rPower_DSP_Produktion 		:= STRING_TO_REAL(fbDSP_Produktion.arrData[7].sValue);                  // Leistung (kW)
	rflow_VL_DSP_Produktion		:= STRING_TO_REAL(fbDSP_Produktion.arrData[3].sValue);					// Temperatur in Grad C
	rflow_RL_DSP_Produktion		:= STRING_TO_REAL(fbDSP_Produktion.arrData[4].sValue);					// Temperatur in Grad C
END_IF

fbHeizkoerper_buero(
	usiAddress 	:= 4,                    	// M-Bus-Adresse(Primär)
	bStart 		:= m_Start4,                // Startflag
	usiUnit     := 1,               		// KW
	bDisabled 	:= FALSE,                 	
	bBusy => , 
	bReady => ,              				// Datenbereit-Status
	bError => , 
	eError => , 
	stCom 		:= stCom
);

IF NOT fbHeizkoerper_buero.bBusy AND fbHeizkoerper_buero.bError THEN

	Err4:= fbHeizkoerper_buero.eError;
END_IF

IF fbHeizkoerper_buero.bReady THEN

    lrEnergy_Heizkoerper_buero 	:= STRING_TO_REAL(fbHeizkoerper_buero.arrData[1].sValue);                 	// Energie (kWh)
    rFlow_Heizkoerper_buero 	:= STRING_TO_REAL(fbHeizkoerper_buero.arrData[6].sValue);                  // Durchfluss (m³/h)
    rPower_Heizkoerper_buero 	:= STRING_TO_REAL(fbHeizkoerper_buero.arrData[7].sValue);                  // Leistung (kW)
	rflow_VL_Heizkoerper_buero	:= STRING_TO_REAL(fbHeizkoerper_buero.arrData[3].sValue);					// Temperatur in Grad C
	rflow_RL_Heizkoerper_buero	:= STRING_TO_REAL(fbHeizkoerper_buero.arrData[4].sValue);					// Temperatur in Grad C
END_IF

fbHalle_Bestand_S100(
	usiAddress 	:= 5,                    	// M-Bus-Adresse(Primär)
	bStart 		:= m_Start5,                // Startflag
	usiUnit     := 1,               		// KW
	bDisabled 	:= FALSE,                 	
	bBusy => , 
	bReady => ,              				// Datenbereit-Status
	bError => , 
	eError => , 
	stCom 		:= stCom
);

IF NOT fbHalle_Bestand_S100.bBusy AND fbHalle_Bestand_S100.bError THEN

	Err5:= fbHalle_Bestand_S100.eError;
END_IF

IF fbHalle_Bestand_S100.bReady THEN

    lrEnergy_Halle_Bestand_S100 	:= STRING_TO_REAL(fbHalle_Bestand_S100.arrData[1].sValue);                 	// Energie (kWh)
    rFlow_Halle_Bestand_S100 		:= STRING_TO_REAL(fbHalle_Bestand_S100.arrData[6].sValue);                  // Durchfluss (m³/h)
    rPower_Halle_Bestand_S100 		:= STRING_TO_REAL(fbHalle_Bestand_S100.arrData[7].sValue);                  // Leistung (kW)
	rflow_VL_Halle_Bestand_S100		:= STRING_TO_REAL(fbHalle_Bestand_S100.arrData[3].sValue);					// Temperatur in Grad C
	rflow_RL_Halle_Bestand_S100		:= STRING_TO_REAL(fbHalle_Bestand_S100.arrData[4].sValue);					// Temperatur in Grad C
END_IF


fbLueftung(
	usiAddress 	:= 6,                    	// M-Bus-Adresse(Primär)
	bStart 		:= m_Start6,                // Startflag
	usiUnit     := 1,               		// KW
	bDisabled 	:= FALSE,                 	
	bBusy => , 
	bReady => ,              				// Datenbereit-Status
	bError => , 
	eError => , 
	stCom 		:= stCom
);

IF NOT fbLueftung.bBusy AND fbLueftung.bError THEN

	Err6:= fbLueftung.eError;
END_IF

IF fbLueftung.bReady THEN

    lrEnergy_Lueftung 	:= STRING_TO_REAL(fbLueftung.arrData[1].sValue);             	// Energie (kWh)
    rFlow_Lueftung 		:= STRING_TO_REAL(fbLueftung.arrData[6].sValue);             	// Durchfluss (m³/h)
    rPower_Lueftung 	:= STRING_TO_REAL(fbLueftung.arrData[7].sValue);            	// Leistung (kW)
	rflow_VL_Lueftung	:= STRING_TO_REAL(fbLueftung.arrData[3].sValue);				// Temperatur in Grad C
	rflow_RL_Lueftung	:= STRING_TO_REAL(fbLueftung.arrData[4].sValue);				// Temperatur in Grad C
END_IF

END_PROGRAM

// ---- POUs/prgComEffIO.TcPOU
PROGRAM prgComEffIO
VAR
	fbCom		: FB_MqttCommunicator_V5;
END_VAR

// CX-7BDACD
fbCom(
	bConnect:= TRUE, 
	strAuthKey := 'ENE87365342998',
	sUserName:= '4a0a6889-c115-4e99-9566-4029ce271fe2', 
	sUserPassword:= 'dd36787c-fc51-4107-9d6e-339f79a51c0d', 
	eSavePositionCertificate:= eSavePositionOnPLC.ePostionHardDisk,
	time_HeartBeat_sec:= T#50S, 
	bConnected=> , 
	bError=> , 
	hrErrorCode=> , 
	eConnectionState=> , 
	eErrorMessage_Out=> );

END_PROGRAM
